// ---- DUTs/METS/Device/Scanner/Hand Scanner/ST_SCANNER_USBConfig.TcDUT
TYPE ST_SCANNER_USBConfig :
STRUCT
	bEnabled					: BOOL;										(* Enable HandScanner *)
	sScannerName				: STRING	:= 'USB';
	bReset					: BOOL;										(* Reset HandScanner *)
	nScannerPosition			: UINT;										(* Array position used in the camera configs.  This allows the HMi to display the handscanner stuff as a microscan camera *)
	sComPort					: STRING(5) := 'COM3';									(* COM port type*)
	nBaudRate				: UINT:= 9600;								(* Baud rate for scanner. 2 = 1200, 3=2400, 4=4800, 5=9600, 6=19200, 7=38400, 8=57600, 9=115200 - Default baudrate for hand sanner sick1910i *)          								 (* 1  *)
	tRXTimeOut				: TIME := T#0ms;
	nPackPerOuter				: INT := 20;
END_STRUCT
END_TYPE

// ---- DUTs/METS/Device/Scanner/NewModel/ST_SCANNER_Ctrl.TcDUT
TYPE ST_SCANNER_Ctrl :    //ST_SCANNER_CameraMap
STRUCT
	bProcessNewCode		: BOOL;
	bTCPTrigger			: BOOL;
	bManualTrigger		: BOOL;
	bResetStats			: BOOL;	
	
	stOptions			: ST_SCANNER_Options;
	stCameraMap			: ST_SCANNER_CtrlMapping;
END_STRUCT
END_TYPE

// ---- DUTs/METS/Device/Scanner/NewModel/ST_SCANNER_CtrlOptions.TcDUT
TYPE ST_SCANNER_CtrlOptions :
STRUCT
	eScannerType			: E_SCANNER_DeviceType;
	nImageBuffer			: INT;
	(*nSequenceProgs		: BYTE;*)
	bUseExternalLight		: BOOL;
	nExpectedResp			: INT;
END_STRUCT
END_TYPE

// ---- DUTs/METS/Device/Scanner/NewModel/ST_SCANNER_IN.TcDUT
TYPE ST_SCANNER_IN :
STRUCT
	stTriggerID				: ST_SCANNER_TriggerID;	(* trigger ID data, will be returned in sImageData to allow trigger and response to be aligned *)
	stManualStatus			: ST_SCANNER_ManualStatus;
	
END_STRUCT
END_TYPE

// ---- DUTs/METS/Device/Scanner/ST_SCANNER.TcDUT
TYPE ST_SCANNER :
STRUCT
	bReady							: BOOL;
	nState							: BYTE;
	bLastBarcodeValid					: BOOL;
(**)	strLastCodeRead					: T_MaxString;
(**)	strLastBarcode						: STRING(253);	(*zenon*)
	strCurrentCodeRead					: T_MaxString;
	aLast10CodesRead					: ARRAY[1..10]  OF T_MaxString;
	strLastStatus						: T_MaxString;
	nTriggerCounter					: UDINT;
	sManualCtrlScanner					: ST_SCANNER_ManualCtrl;
(**)(*	sSStats							: ST_SCANNER_Statistics;*)
	sScannerOpState					: ST_SCANNER_OpState;
	sImageData						: ST_SCANNER_ImageData;
	bEnableActive						: BOOL;
	nActiveProgram					: BYTE;
	bAcceptTrigger						: BOOL;
	sTriggerID							: ST_SCANNER_TriggerID;
	eSocketState						: E_SocketConnectionState;
	sReadPerformance					: ST_SCANNER_Performance;
END_STRUCT
END_TYPE

// ---- DUTs/METS/Device/Scanner/ST_SCANNER_ApplicationIdentifier.TcDUT
TYPE ST_SCANNER_ApplicationIdentifier :
STRUCT
	strAI		: STRING(4);
	bFixed		: BOOL;
	nLength		: UINT;
END_STRUCT
END_TYPE

// ---- DUTs/METS/Device/Scanner/ST_SCANNER_CameraMap.TcDUT
TYPE ST_SCANNER_CameraMap :
STRUCT
	nIndex				: INT;
	nReqProgram			: BYTE;
	stOptions				: ST_SCANNER_Options;
	aPackPos				: ARRAY[1..5, 1..cMAX_CAMERA_PROG_NUMBER] OF BYTE;
	aTargetBuffer			: ARRAY[1..5] OF BYTE;

END_STRUCT
END_TYPE

// ---- DUTs/METS/Device/Scanner/ST_SCANNER_CodeData.TcDUT
TYPE ST_SCANNER_CodeData :
STRUCT
	nScannerIndex			: INT;			(* scanner index when an array of scanners is used *)
	strDataString			: T_MaxString;	(* data string read from code *)
	eCodeType			: E_SCANNER_CodeType;	(* code type *)
	fOverallGrade			: LREAL;		(* overall grade of code *)
	fXPos				: LREAL;		(* X position of centre of code *)
	fYPos				: LREAL;		(* Y position of centre of code *)
	fAngle				: LREAL;		(* angle of code *)
	fCellSize				: LREAL;		(* cell size *)
	fSymbolContrast		: LREAL;		(* symbol contrast *)
	nEvaluation			: INT;			(* general code quality evaluatio*)
	fUnusedErrCorr			: LREAL;		(* unused error correction *)
	nProgramNo			: BYTE;			(* program number *)
END_STRUCT
END_TYPE

// ---- DUTs/METS/Device/Scanner/ST_SCANNER_Config.TcDUT
TYPE ST_SCANNER_Config :
STRUCT
	sDeviceName				: STRING(30) := 'Camera';
	bDisableCameraUse		: BOOL;
	aCameraWarningLevel		: INT := 90;
	stCameraIP					: ST_TCPIP_AddressPort;
	tTimeOut					: TIME := t#3s;
	eCameraVendor			: E_SCANNER_Vendor;
	bDontParseAsGS1			: BOOL;

	eScannerType			: E_SCANNER_DeviceType;
	eExpectedType			: E_SCANNER_CodeType;
	bUseExternalLight		: BOOL;
	nLightingIntensity		: INT;
	nDisplayDelayConfig	: BOOL;

	nImageBuffer			: INT := 1;
	nExpectedResp			: INT := 1;
END_STRUCT
END_TYPE

// ---- DUTs/METS/Device/Scanner/ST_SCANNER_Evaluation.TcDUT
TYPE ST_SCANNER_Evaluation :
STRUCT
	nTotalReads			: UDINT;
	nReadCodes			: UDINT;
	nNOKCodes			: UDINT;

	nGoodCodes			: UDINT;
	nFairCodes			: UDINT;
	nPoorCodes			: UDINT;

	fReadEfficiency			: LREAL;
	fNOKEfficiency			: LREAL;

	fGoodEfficiency		: LREAL;
	fFairEfficiency			: LREAL;
	fPoorEfficiency			: LREAL;

END_STRUCT
END_TYPE

// ---- DUTs/METS/Device/Scanner/ST_SCANNER_ImageData.TcDUT
TYPE ST_SCANNER_ImageData :
STRUCT
	nCodesRead		: INT;
	tScanTime		: TIME;		(* image cycle time (including image acquisition time and decode time) *)
	sStatus			: T_MaxString;
	stTriggerID		: ST_SCANNER_TriggerID;
	aCodeData		: ARRAY[1..cMAX_CAMERA_PROG_NUMBER] OF ST_SCANNER_CodeData;
END_STRUCT
END_TYPE

// ---- DUTs/METS/Device/Scanner/ST_SCANNER_ManualCtrl.TcDUT
TYPE ST_SCANNER_ManualCtrl :
STRUCT
	bManualTrigger		: BOOL;		(*zenon*)
	bConfigure			: BOOL;		(*zenon*)
	bBrowseLive			: BOOL;		(*zenon*)
	bBrowseDiag			: BOOL;		(*zenon*)
	bResetStats			: BOOL;		(*zenon*)
END_STRUCT
END_TYPE

// ---- DUTs/METS/Device/Scanner/ST_SCANNER_OpState.TcDUT
TYPE ST_SCANNER_OpState :
STRUCT
	bReady				: BOOL;
	nActiveProgram		: BYTE;
	bAcceptTrigger		: BOOL;
	bCodeChangeActive	: BOOL;
	nActiveTriggers		: INT;
	nExpectedResp			: INT;
	tAcquisitionTime	: TIME;
	nStatusByte			: BYTE;
	nErrorCode			: UDINT;
	nOpState			: BYTE;
END_STRUCT
END_TYPE

// ---- DUTs/METS/Device/Scanner/ST_SCANNER_Options.TcDUT
TYPE ST_SCANNER_Options :
STRUCT
	eScannerType			: E_SCANNER_DeviceType;
	nImageBuffer			: INT;
	(*nSequenceProgs		: BYTE;*)
	bUseExternalLight		: BOOL;
	nExpectedResp			: INT;
END_STRUCT
END_TYPE

// ---- DUTs/METS/Device/Scanner/ST_SCANNER_Performance.TcDUT
TYPE ST_SCANNER_Performance :
STRUCT
	tLastDiff : TIME;
	tAverageDiff : TIME;
	arrTimeDiff : ARRAY[0..9] OF TIME;
END_STRUCT
END_TYPE

// ---- DUTs/METS/Device/Scanner/ST_SCANNER_Statistics.TcDUT
TYPE ST_SCANNER_Statistics :
STRUCT
	nTotalReads			: UDINT;
	nValidCodes			: UDINT;
	nInvalidCodes			: UDINT;
	nDuplicateCodes		: UDINT;
	nNoCodeFound		: UDINT;
END_STRUCT
END_TYPE

// ---- DUTs/METS/Device/Scanner/ST_SCANNER_TriggerID.TcDUT
TYPE ST_SCANNER_TriggerID :
STRUCT
	nTriggerID			: UDINT;
	nScanNo				: INT := 1;
	nScannerIndex		: INT := 1;
END_STRUCT
END_TYPE

// ---- DUTs/METS/Files/E_FILE_CtrlState.TcDUT
TYPE E_FILE_CtrlState :
(
	E_CX_FILEIDLE,
	E_CX_FILEOPEN,
	E_CX_FILESEEK,
	E_CX_FILEREAD,
	E_CX_FILEWRITE,
	E_CX_FILECLOSE,
	E_CX_FILEDONE
);
END_TYPE

// ---- DUTs/METS/Files/E_FILE_DeleteOldFilesState.TcDUT
TYPE E_FILE_DeleteOldFilesState :
(
	E_OLDFILE_IDLE,
	E_OLDFILE_CURRENTTIME,
	E_OLDFILE_FILELIST1,
	E_OLDFILE_DELETEFILELIST1,
	E_OLDFILE_FILELIST2,
	E_OLDFILE_DELETEFILELIST2,
	E_OLDFILE_ABORTFILELIST,
	E_OLDFILE_FINDFOLDER,
	E_OLDFILE_FINDFILE,
	E_OLDFILE_DELETEFOLDER,
	E_OLDFILE_DELETEFILE,
	E_OLDFILE_DONE
);
END_TYPE

// ---- DUTs/METS/Files/E_FILE_State.TcDUT
TYPE E_FILE_State :
(
	E_FILE_IDLE,
	E_FILE_GETSIZE,
	E_FILE_OPEN,
	E_FILE_OPEN2,
	E_FILE_READ,
	E_FILE_READ2,
	E_FILE_WRITE,
	E_FILE_CLOSE,
	E_FILE_CLOSE2,
	E_FILE_COPY,
	E_FILE_COMPARE,
	E_FILE_ABORT,
	E_FILE_DELETE,
	E_FILE_MOVE,
	E_FILE_CHECKIFEXISTS,
	E_FILE_SEEK,
	E_FILE_FINDFILE,
	E_FILE_NEXTFILE,
	E_FILE_CLOSELIST,
	E_FILE_DONE
);
END_TYPE

// ---- DUTs/METS/Files/ST_FILE_WriteFileStatistic.TcDUT
TYPE ST_FILE_WriteFileStatistic :
STRUCT
	nTotalFilesWritten				: UDINT;
	nGoodFilesWritten				: UDINT;
	nBadFilesWritten				: UDINT;
	nFileWriteErrors				: UDINT;

	nTotalFilesVerified				: UDINT;
	nEmptyFilesVerified				: UDINT;
	nSizeErrorsVerified				: UDINT;
	nGoodFilesVerified				: UDINT;
	nFileVerifyNotFound			: UDINT;
	nFileVerifyErrors				: UDINT;
END_STRUCT
END_TYPE

// ---- DUTs/METS/HMI/Device Manual Control/ST_HMI_AxisCtrl.TcDUT
TYPE ST_HMI_AxisCtrl :
STRUCT
	stReqEanble		: ST_HMI_Buttons;
	stReqReset		: ST_HMI_Buttons;
	stReqPositioning	: ST_HMI_Buttons;	(*Button start positioning manual mode*)
	stRelease			: ST_HMI_Buttons;

	stReqJogFwd			: ST_HMI_Buttons;		(* set TRUE to jog forwards *)
	stReqJogRev			: ST_HMI_Buttons;		(* set TRUE to jog reverse *)
	fJogVelocity			: LREAL;	(* jog velocity (does not take effect if jog is in progress *)

	eMotionType		: E_AXIS_MotionType;

	fDistance			: LREAL;	(*target relative position*)
	fPosition			: LREAL;	(*target absolute position*)
	fVelocity			: LREAL;	(* target velocity *)
	bStopAtPos		: BOOL;	(* set TRUE to stop at specified pos, set FALSE to stop immediately *)
	fStopPos			: LREAL;	(* target modulo stop position *)

	(*eMotionState 		: MC_AxisStates;*)

END_STRUCT
END_TYPE

// ---- DUTs/METS/HMI/Device Manual Control/ST_HMI_G120Ctrl.TcDUT
TYPE ST_HMI_G120Ctrl :
STRUCT
	stRun				: ST_HMI_Buttons;
	stReset				: ST_HMI_Buttons;
	nSpeedHz 			: UINT;
	stInvertDirection	: ST_HMI_Buttons;
END_STRUCT
END_TYPE

// ---- DUTs/METS/HMI/Device Manual Control/ST_HMI_PrinterCtrl.TcDUT
TYPE ST_HMI_PrinterCtrl :
STRUCT
	stPrinterSelect		: ST_HMI_Buttons;
	stPrintLabel		: ST_HMI_Buttons;
	stApplyLabel		: ST_HMI_Buttons;	(*Button start positioning manual mode*)
	stPrinterReset		: ST_HMI_Buttons;

END_STRUCT
END_TYPE

// ---- DUTs/METS/HMI/Device Status/E_HMI_DriveStatus.TcDUT
TYPE E_HMI_DriveStatus :
(
	E_DRIVE_UNKNOWN := 0,
	E_DRIVE_SPOPPED := 1,
	E_DRIVE_RUNING := 2,
	E_DRIVE_ERROR := 3
);
END_TYPE

// ---- DUTs/METS/HMI/Device Status/ST_HMI_AxisStatus.TcDUT
//{warning 'CONVERSION MESSAGE: This text contained unprintable characters, that have been deleted'.}
TYPE ST_HMI_AxisStatus :
STRUCT

(* read only *)

	eMotionState 		: MC_AxisStates;

	bInitOK				: BOOL;
	bEnabled			: BOOL;
	bHomeActive			: BOOL;
	bVeloActive			: BOOL;
	bRelativeActive		: BOOL;
	bAbsoluteActive		: BOOL;
	bJogActive			: BOOL;


	bOperational 				: BOOL;
	bHasJob						: BOOL;
	bInTargetPosition 			: BOOL;
	bInPositionRange 			: BOOL;
	bHomed 						: BOOL;
	bHomingBusy 				: BOOL;
	bMovingPositiveDirection 	: BOOL;
	bMovingNegativeDirection	: BOOL;
	bNotMoving 					: BOOL;

	bError 						: BOOL;
	nErrorId 					: UDINT;

	fActualPosition 			: LREAL;
	fActualVelocity 			: LREAL;
	fSetpointPosition 			: LREAL;


END_STRUCT
END_TYPE

// ---- DUTs/METS/HMI/Device Status/ST_HMI_CylinderStatus.TcDUT
TYPE ST_HMI_CylinderStatus :
STRUCT

(* read only *)
	bDeviceDisable			: BOOL;
	bMoveNotAllowed			: BOOL;

	bErrorPosition				: BOOL;
	bInPosition				: BOOL;
	bHomePosition				: BOOL;

	bCylinderInRetractedPosition	: BOOL;
	bCylinderInExtendedPosition	: BOOL;
	bCylinderIsRetracting		: BOOL;
	bCylinderIsExtending		: BOOL;

	stTagID					: ST_CYLINDER_TagID;

END_STRUCT
END_TYPE

// ---- DUTs/METS/HMI/Device Status/ST_HMI_HoneywellStatus.TcDUT
TYPE ST_HMI_HoneywellStatus :
STRUCT

(* read only *)
	bHandScanerPortOK			: BOOL;
	bHandScannerBaudrateOK	: BOOL;
	sLastScannerBarcode		: T_MaxString;

END_STRUCT
END_TYPE

// ---- DUTs/METS/HMI/Device Status/ST_HMI_PrinterStatus.TcDUT
TYPE ST_HMI_PrinterStatus :
STRUCT
	sPrinterName					: STRING(30);
(* read only *)
	bPrinterReady					: BOOL;
	bActivePrinter					: BOOL;
	bPrinterInService				: BOOL;		(*printer Avalable*)
	bPrinterSelected				: BOOL;
	bDataReady					: BOOL;
	bHomePosition				: BOOL;
	bLabelPrinted					: BOOL;
	bReadyToApply				: BOOL;
	bApplyDone					: BOOL;
	bSummaryWarning				: BOOL;
	bPrinterError					: BOOL;

	Q								: ST_PRINTER_OUT;

END_STRUCT
END_TYPE

// ---- DUTs/METS/HMI/HMIQueue/ST_HMI_CAC_Data.TcDUT
TYPE ST_HMI_CAC_Data :
STRUCT
	sBarcode 				: T_CASE_Barcode;
	(*sCaseIDCode			: STRING(10);
	sProductionDate			: STRING(10);
	sProductionTime			: STRING(8);
	sCaseRejectCode			: T_MaxString;		(* blank and not included in CAC files for valid cases *)*)
	nNumberOfOuters			: INT;
	nNumberOfPacks			: INT;
	aOuter					: ARRAY[1..cMAX_HMI_OUTERS_PER_CASE] OF ST_HMI_OAC_Data;
END_STRUCT
END_TYPE

// ---- DUTs/METS/HMI/HMIQueue/ST_HMI_CaseVerifiedCode.TcDUT
TYPE ST_HMI_CaseVerifiedCode :
STRUCT
	sCaseIDCode				: STRING(10);
	sProductionDate			: STRING(10);
	sProductionTime			: STRING(8);
END_STRUCT
END_TYPE

// ---- DUTs/METS/HMI/HMIQueue/ST_HMI_CASE_CaseQueue.TcDUT
TYPE ST_HMI_CASE_CaseQueue :
STRUCT
	aCACData		: ARRAY[1..cMAX_CASE_QUEUE] OF ST_HMI_CAC_Data;	(* array of CAC data *)
END_STRUCT
END_TYPE

// ---- DUTs/METS/HMI/HMIQueue/ST_HMI_OAC_Data.TcDUT
TYPE ST_HMI_OAC_Data :
STRUCT
	sBarcode				: T_OUTER_Barcode;
	aPackCode				: ARRAY[1..cMAX_HMI_PACKS_PER_OUTER] OF T_HMI_PACK_Barcode;
END_STRUCT
END_TYPE

// ---- DUTs/METS/HMI/HMIQueue/ST_HMI_OCV_Data.TcDUT
TYPE ST_HMI_OCV_Data :
STRUCT
	sPackCode			: T_PACK_Barcode;
	nPackStatus		: BYTE;
END_STRUCT
END_TYPE

// ---- DUTs/METS/HMI/HMIQueue/ST_HMI_OuterStatus.TcDUT
TYPE ST_HMI_OuterStatus :
STRUCT
	sBarcode						: T_OUTER_Barcode;

	sOuterRejectCode				:  T_RejectCode;
	nOuterRejectID					:  UINT;

	aAggregationCodes			: ARRAY[1..2] OF T_PACK_Barcode;
	aAggregationCodesPosition	: ARRAY[1..2] OF INT;

	aPackRejectCode				: ARRAY[1..cMAX_HMI_PACKS_PER_OUTER] OF T_RejectCode;
	aPackRejectID					: ARRAY[1..cMAX_HMI_PACKS_PER_OUTER] OF INT;

	sProductionDate				: STRING(10);
	sProductionTime				: STRING(8);

	aPackCode						: ARRAY[1..cMAX_HMI_PACKS_PER_OUTER] OF T_PACK_Barcode;
	aOACPackStatus				: ARRAY[1..cMAX_HMI_PACKS_PER_OUTER] OF BYTE;	(* OAC pack code status *)

	nNumberOfPacks				: INT;
	nAcceptanceLevel				: INT;
	nNumberOfLinkedPacks		: INT;
	nMaxOuterStatusQueue		: INT;

END_STRUCT
END_TYPE

// ---- DUTs/METS/HMI/HMIQueue/ST_HMI_PLAS_Queue.TcDUT
TYPE ST_HMI_PLAS_Queue :
STRUCT
(*Pack Infeed queue*)
	nInfeedIndex					: INT;				(* number of Outers in queue *)
	aPackInfeedQueue				: ARRAY[1..cMAX_HMI_PACK_INFEED_QUEUE] OF T_HMI_PACK_Barcode; (* pack infeed queue + status (999)*)

(*Pack Buffer intermediat queue*)
	aBufferQueue					: ARRAY[1..cMAX_HMI_PACK_INFEED_QUEUE] OF T_HMI_PACK_Barcode; (* intermediat pack queue + status (999)*)

(*OCV Data*)
	sProductionDate				: STRING(10);
	sProductionTime				: STRING(8);

	aOCVData						: ARRAY[1..cMAX_HMI_PACKS_PER_OUTER] OF T_HMI_PACK_Barcode; (* pack queue + status (999)*)

	nNumberOfPacks				: INT;
	nAcceptanceLevel				: INT;
	nNumberOfLinkedPacks		: INT;
	nMaxPackPerOuter				: INT; (*real number of codes*)

END_STRUCT
END_TYPE

// ---- DUTs/METS/HMI/ST_HMI_Buttons.TcDUT
TYPE ST_HMI_Buttons :
STRUCT

	bButtonState			: 	BOOL;
	bButtonRisingEdge		:	BOOL;
   	bButtonFallingEdge		:	BOOL;
	(*nChangeLogID			: 	INT;*)


(*	bStartButtonRisingEdge		:	BOOL;
   	bStartButtonFallingEdge		:	BOOL;
    	bResetButtonRisingEdge		:	BOOL;
    	bResetButtonFallingEdge		:	BOOL;
    	bStopButtonRisingEdge		:	BOOL;
    	bStopButtonFallingEdge		:	BOOL;*)
END_STRUCT
END_TYPE

// ---- DUTs/METS/HMI/ST_HMI_StationStatus.TcDUT
TYPE ST_HMI_StationStatus :
STRUCT

	bSeqAbort					: BOOL;		(**)
	bSeqIsHoming				: BOOL;
	bSeqInProgress				: BOOL;		(**)
	bSeqComplete				: BOOL;		(**)
	bSeqError					: BOOL;
	nSeqErrorID					: UDINT;

	bStationHomed				: BOOL;		(**)
	bStationNotMoving			: BOOL;		(**)



END_STRUCT
END_TYPE

// ---- DUTs/METS/HMI/ST_HMI_Visualisation.TcDUT
TYPE ST_HMI_Visualisation:
STRUCT
	(*Test outputs*)
(*	bEnableForcingOutputs			: BOOL;

	bForceEUCAMachineRun_STCP		: BOOL;	(*to set qb82KF1_1_EUCAMachineRun*)
	bForceCaseValidationOK_STCP		: BOOL;	(*to set qb82KF1_5_CaseValidationOK*)
	bForceOuterValidationOK_STCP	: BOOL;	(*to set qb82KF1_2_OuterValidationOK*)
	bForceLabellerInhibit_STL		: BOOL;	(*to set qb82KF1_3_LabellerInhibit_STL*)
	bForceTPDMachineRun			: BOOL;	(*to set qb482KF1_4_TPDMachineRun*)
	bForceSpare					: BOOL;
*)

	(*Update PCM*)
	bEnableUpdatePCM				: BOOL;

	strLastRetailSKU 				: T_CodeRSKU;
	strLastProductionOrder			: T_CodePO;
	strLastBatchNumber				: T_CodeBATCH;

	strLastPackGTIN 				: T_CodeGTIN;
	strLastOuterGTIN 				: T_CodeGTIN;
	strLastCaseGTIN 				: T_CodeGTIN;

END_STRUCT
END_TYPE

// ---- DUTs/METS/KPI/ST_KPI_CasePackerSignals.TcDUT
TYPE ST_KPI_CasePackerSignals :
STRUCT
	nSensor			: UDINT;
	nMachine		: UDINT;
	nPLC			: UDINT;

END_STRUCT
END_TYPE

// ---- DUTs/METS/KPI/ST_KPI_CodePos.TcDUT
TYPE ST_KPI_CodePos :
STRUCT
	ReadOK				: UDINT;
	Efficiency			: LREAL;
END_STRUCT
END_TYPE

// ---- DUTs/METS/KPI/ST_KPI_InspectionEfficency.TcDUT
TYPE ST_KPI_InspectionEfficency :
STRUCT
	ProcessedTotal			: UDINT;
	ProcessedSuccessful		: UDINT;
	ProcessedRejected		: UDINT;
	ProcessedEfficiency		: LREAL;
END_STRUCT
END_TYPE

// ---- DUTs/METS/KPI/ST_KPI_ItemsProduced.TcDUT
TYPE ST_KPI_ItemsProduced :
STRUCT
	Total					: UDINT;
	Passed				: UDINT;
	Rejected				: UDINT;
	Efficiency				: LREAL;
	CreatedFiles			: UDINT;
	WarningLevel			: REAL := 99.75;
	AlarmLevel			: REAL := 99.50;
END_STRUCT
END_TYPE

// ---- DUTs/METS/KPI/ST_KPI_OCVFile.TcDUT
TYPE ST_KPI_OCVFile :
STRUCT
	nOCVFiles					: UDINT;
	nOuterStoredInOCV				: UDINT;
	nLinkedPackInOCV				: UDINT;
	nOCVWriteErrorCounter			: UDINT;
END_STRUCT
END_TYPE

// ---- DUTs/METS/KPI/ST_KPI_OutersProcessing.TcDUT
TYPE ST_KPI_OutersProcessing :
STRUCT
	AtPackAggregCameras	: UDINT;
	AtConfimrationCamera 	: UDINT;
	AtValidationCamera		: UDINT;
END_STRUCT
END_TYPE

// ---- DUTs/METS/KPI/ST_KPI_OutersProduced.TcDUT
TYPE ST_KPI_OutersProduced :
STRUCT
	Total					: UDINT;
	Passed				: UDINT;
	Rejected				: UDINT;
	Efficiency				: LREAL;
END_STRUCT
END_TYPE

// ---- DUTs/METS/LogData/E_LOG_Handler.TcDUT
{attribute 'qualified_only'}
TYPE E_LOG_Handler :
(
	
(**************** Keep in mind limited number of E_NUM elements (array of FB handlers) fixed size to 256 ******************)
		
(* FSS connection logs *)
		OKCONECCTIONTOFSS,
		LOSTCONECCTIONTOFSS,
		
		(* Doors logs*)
		DOOROPENZONE1,
		DOOROPENZONE2,
		MASTERLISTDOOR,
		AGGREGATIONDOOR,
		PACKWRAPPERDOOR,
		
(* Control buttons logs*)
		STARTBUTTONPRESSED,
		STOPBUTTONPRESSED,
		RESETBUTTONPRESSED,
		
(* Machines not running status logs *)
		EUCANOTRUNNINGPT,
		EUCANOTRUNNINGCT,
		TPDNOTRUNNINGPT,
		TPDNOTRUNNINGCT,	
		EXTNOTRUNNINGPT,
		EXTNOTRUNNINGCT,
		
(* Machines state changed *)
		MACHINESTATEPT,
		MACHINESTATECT,
		
(**************** PACK AGGREGATION MODE ****************)		
		
(*PAOL SEQUENCE - 2CAM_METSONE*)				
		PAOL2CAMPACKAGGTRIG,		
		PAOL2CAMCAM1,		
		PAOL2CAMCAM2,
		PAOL2CAMPA1ADDED,
		PAOL2CAMPA2ADDED,	
		
(*PAOL SEQUENCE - 3CAM_LIHTBOX*)
		PAOL3CAMPA1ADDED,		
		PAOL3CAMPA2ADDED,
		PAOL3CAMPA3ADDED,
		
(*PLAS SEQUENCE - T01*)
		T01CAMAGG1,
		T01CAMAGG2,		
		T01CAMAGGTRIG,
		T01STACKERTRIG,
		T01AGGITEM,
		T01AGGADDED,
		T01WRAPPER1REJECT,
				
(*PLAS SEQUENCE - T02*)
		T02CAMAGG1,
		T02CAMAGG2,
		T02CAMAGGTRIG,
		T02STACKERTRIG,
		T02CAMINTERTRIG,
		T02CAMINTER,
		T02INTERQUEUE,
		T02AGGITEM,
		T02AGGADDED,
		T02WRAPPER1REJECT,
		
(*PLAS SEQUENCE - T03*)
		T03CAMAGG,
		T03CAMAGGTRIG,
		T03CAMCONFTRIG,
		T03CAMINTERTRIG,
		T03CAMINTER,
		T03INTERQUEUE,
		T03CAMCON,
		T03PACKINDEX,
		T03MOVEDTOOCV,
		T03WRAPPERREJECT,
		
(*PLAS SEQUENCE - T04*)		
		T04CAMAGG,
		T04CAMAGGTRIG,	
		T04CAMCONFTRIG,
		T04CAMINTERTRIG,
		T04CAMINTER,
		T04INTERQUEUE,
		T04CAMCON,
		T04PACKINDEX,
		T04MOVEDTOOCV,
		T04WRAPPERREJECT,
		
(**************** PACK AGGREGATION MODE ****************)
		
(* OCV logs *)
		STACKOUTOFSEQ,
		LASTOCVCONTENT,
		
(* OAC logs *)
		LASTOACCONTENT,
		
(* Printers comands *)
		LASTPRINTER01COMMAND,
		LASTPRINTER02COMMAND,
		LASTPRINTER03COMMAND,
		LASTPRINTER04COMMAND,
		LASTPRINTER05COMMAND,
		LASTPRINTER06COMMAND,
		
(* Case Packer Sequence logs *)
		OUTERCOMPLETE,
		ROWCOMPLETE,
		LAYERCOMPLETE,
		INTERMEDIATECOMPLETE,
		CASECOMPLETE,		
		CASEDISCHARGERT,
		CASEDISCHARGEFT,
		CASELABELVALIDATION,
		
(* Cameras timeout logs *)
		OUTERAGGREGATIONCODE,
		
(* Data move/handeling status logs*)
		ROWCOMPLETECODES,
		LAYERCOMPLETECODES,
		FINALISECASECONTENTCODES,
		
(* Data LogIn DB logs*) (* NOT INTUITIVE NAMES - to be changed ?? *)
		INTERPUSHOVERWIRTTEN,
		CASECOMPLETEOVERWITTEN,
		CASEDISCHARGEOVERWRITTEN,
		
(* Rejects handling logs *)
		REJECTEDBYCASEPACKER,
		
(* Case events logs *)
		CASELABELCODE,
		MCCREATEDEVENT,
		CASEVALIDATIONRT,
		CASEVALIDATIONFT,
		
(* Data files write error logs *)
		OCVWRITEERROR,
		OACWRITEERROR,
		CACWRITEERROR,
		CHMWRITEERROR,
		
(* Master List status logs *)
		MLFILLINSTATUS,
		MLSTATUS,
		MLRESOTRESTATUS,
		//E_LOG_WRAPPERREJECT1,
		WRAPPERREJECT2
		
);
END_TYPE

// ---- DUTs/METS/LogData/ST_LOG_Alarms.TcDUT
TYPE ST_LOG_Alarms :
STRUCT

	nAlarmCounter				: UINT;
	sTotalAlarmTime				: T_TimeLog;
	sMaxAlarmTime				: T_TimeLog;
	stMaxAlarmTimeStamp			: TIMESTRUCT;

END_STRUCT
END_TYPE

// ---- DUTs/METS/LogData/ST_LOG_EventData.TcDUT
TYPE ST_LOG_EventData :
STRUCT
	bEnable					: BOOL;
	nCounter				: UDINT;
	sTimeStamp				: STRING;
	nImageByte				: UINT;
	aDataLogImage			: ARRAY[0..65000] OF BYTE;
	nMaxImageArraySize		: UINT := 65000 ;
	nControlSize			: UINT;
	bBufferOverflow			: BOOL;
END_STRUCT
END_TYPE

// ---- DUTs/METS/LogData/ST_LOG_FileWriteError.TcDUT
TYPE ST_LOG_FileWriteError :
STRUCT
	nWriteErrorID			: UDINT;
	sTimeStamp				: STRING;
	strFileName				: T_MaxString;
END_STRUCT
END_TYPE

// ---- DUTs/METS/LogData/ST_LOG_MachineState.TcDUT
TYPE ST_LOG_MachineState :
STRUCT

	sPowerUp					: T_TimeLog;
	sImmediateStopped			: T_TimeLog;
	sMachineInError				: T_TimeLog;
	sSystemInitialising			: T_TimeLog;
	sSystemManual				: T_TimeLog;
	sSystemReadytoStart			: T_TimeLog;
	sStopping					: T_TimeLog;
	sSystemRunning				: T_TimeLog;
	sMachineWaitingForProduct	: T_TimeLog;
	sConveyorModeActive			: T_TimeLog;
	sSystemConditionalRunning	: T_TimeLog;

END_STRUCT
END_TYPE

// ---- DUTs/METS/LogData/ST_LOG_WriteImageData.TcDUT
TYPE ST_LOG_WriteImageData :
STRUCT
	aLogPT			: ARRAY[0..65000] OF BYTE;
	aLogML			: ARRAY[0..65000] OF BYTE;
	aLogOT			: ARRAY[0..65000] OF BYTE;
	aLogCT			: ARRAY[0..65000] OF BYTE;
END_STRUCT
END_TYPE

// ---- DUTs/METS/NV Data/ST_NOVRAM_METS_Cameras.TcDUT
TYPE ST_NOVRAM_METS_Cameras :
STRUCT
	MachineID					: ST_SYSTEM_MachineID;
	StartDateTime					: T_ISO8601Time;
	CodingAndTrackingMode			: INT;

	aCameraEvaluation				: ARRAY[1..cMAX_CAMERA_NUMBER] OF ST_SCANNER_Evaluation;

	(*CameraPackEval				: ARRAY[1..6] OF ST_SCANNER_Evaluation;
	CameraConfirmEval				: ARRAY[1..2] OF ST_SCANNER_Evaluation;
	CameraOuterValidEval			: ST_SCANNER_Evaluation;
	CameraOuterAggregEval			: ST_SCANNER_Evaluation;
	CameraCaseContentEval			: ST_SCANNER_Evaluation;
	CameraCaseLableEval			: ST_SCANNER_Evaluation;*)

END_STRUCT
END_TYPE

// ---- DUTs/METS/NV Data/ST_NOVRAM_METS_CaseInspactionLog.TcDUT
TYPE ST_NOVRAM_METS_CaseInspactionLog :
STRUCT

	MachineID						: ST_SYSTEM_MachineID;
	StartDateTime						: T_ISO8601Time;
	CodingAndTrackingMode				: INT;
	nPacksPerCase						: INT;			(* Amount Of  Packs per Case unit for current PCM *)
	nOutersPerCase					: INT;

	(*infeed conveyer*)
	nOuterProcessed					: UDINT;
	nOuterAggregated					: UDINT;
	nMasterListRestoredSuccessful		: UDINT;
	nMasterListRemoved				: UDINT;
	nQualityRejects					: UDINT;

	(*row validation*)
	nRowValidationIndexUnder			: UDINT;
	nRowValidationIndexOver			: UDINT;
	nRowValidationIndexCorrect			: UDINT;
	nRowValidationIndexNotFound		: UDINT;

	(*outer to case validation*)
	nOuterToCaseValidationIndexUnder		: UDINT;
	nOuterToCaseValidationIndexOver		: UDINT;
	nOuterToCaseValidationIndexCorrect	: UDINT;
	nOuterToCaseValidationIndexNoData	: UDINT;

	(*case validation*)
	nCaseValidationScanned				: UDINT;
	nCaseValidationCorrect				: UDINT;
	nCaseValidationCasePackerReject		: UDINT;
	nCaseValidationNoCaseLabel			: UDINT;


END_STRUCT
END_TYPE

// ---- DUTs/METS/NV Data/ST_NOVRAM_METS_DualInputs.TcDUT
TYPE ST_NOVRAM_METS_DualInputs :
STRUCT

	MachineID					: ST_SYSTEM_MachineID;
	StartDateTime					: T_ISO8601Time;
	CodingAndTrackingMode			: INT;

	RowComplete			:	ST_KPI_CasePackerSignals;
	LayerComplete			:	ST_KPI_CasePackerSignals;
	CaseComplete			:	ST_KPI_CasePackerSignals;
	CaseDischarged		:	ST_KPI_CasePackerSignals;
	CaseLabelValidation		:	ST_KPI_CasePackerSignals;


END_STRUCT
END_TYPE

// ---- DUTs/METS/NV Data/ST_NOVRAM_METS_Inspection.TcDUT
TYPE ST_NOVRAM_METS_Inspection :
STRUCT
	MachineID					: ST_SYSTEM_MachineID;
	StartDateTime					: T_ISO8601Time;
	CodingAndTrackingMode			: INT;
	AcceptanceLevel				: INT;
	PacksPerOuter					: INT;
	OutersProcessing				: ST_KPI_OutersProcessing;
	OCVFileEfficiency				: ST_KPI_OCVFile;

	PacksRead					: ARRAY[0..cMAX_PACKS_PER_OUTER] OF UDINT;
	PackPosEfficiency				: ARRAY[1..cMAX_PACKS_PER_OUTER] OF ST_KPI_CodePos;

	PackAggregationEfficiency		: ST_KPI_InspectionEfficency;
	PackProduced					: ST_KPI_ItemsProduced;

	aConfirmCodeEfficiency			: ARRAY[1..2] OF ST_KPI_CodePos;
	PackConfirmationEfficiency		: ST_KPI_InspectionEfficency;
	aValidCodeEfficiency			: ARRAY[1..2] OF ST_KPI_CodePos;
	OuterValidationEfficiency			: ST_KPI_InspectionEfficency;

	OuterAggregationEfficiency		: ST_KPI_InspectionEfficency;
	OutersProduced				: ST_KPI_ItemsProduced;

	(*CaseContentValidEfficiency		: ST_KPI_InspectionEfficency;
	CaseLableValidEfficiency			: ST_KPI_InspectionEfficency;*)

	CaseAggregationEfficiency		: ST_KPI_InspectionEfficency;
	CaseProduced					: ST_KPI_ItemsProduced;


END_STRUCT
END_TYPE

// ---- DUTs/METS/Outers/E_OUTER_AgrregationState.TcDUT
TYPE E_OUTER_AgrregationState :
(
	E_OUTER_IDLE_OCV,
	E_OUTER_READ_OCV,
	E_OUTER_ERROR_OCV_READ,
	E_OUTER_BUILD_OAC_DATA,
	E_OUTER_DONE_OCV
);
END_TYPE

// ---- DUTs/METS/Outers/E_OUTER_State.TcDUT
TYPE E_OUTER_State :
(
	E_OUTER_IDLE,
	E_OUTER_SCAN,
	E_OUTER_VALIDATE,
	E_OUTER_CHECKPACKS,
	E_OUTER_KPI,
	E_OUTER_STATUS,
	E_OUTER_DBREQUEST,
	E_OUTER_DBRESPONSE,
	E_OUTER_BUILDXMLIMAGE,
	E_OUTER_WRITEXMLIMAGE,
	E_OUTER_WRITESECONDXMLIMAGE,
	E_OUTER_CREATEERRORFOLDER,
	E_OUTER_UPDATEDATA,
	E_OUTER_WRITEDATA,
	E_OUTER_DELETEFILE,
	E_OUTER_UPDATESTATUS,
	E_OUTER_FINDFILE,
	E_OUTER_READDATA,
	E_OUTER_UPDATEINFEEDQUEUE,
	E_OUTER_DELETECONVQUEUE,
	E_OUTER_DONE
);
END_TYPE

// ---- DUTs/METS/Outers/OAC/E_OAC_State.TcDUT
TYPE E_OAC_State :
(
	E_OAC_IDLE,
	E_OAC_HEADER,
	E_OAC_PACKDATA,
	E_OAC_MOVENAS,
	E_OAC_MOVELOCAL,
	E_OAC_VALIDATEOUTER,
	E_OAC_VALIDATEPACK,
	E_OAC_DBREQUEST,
	E_OAC_DBRESPONSE,
	E_OAC_READFILE,
	E_OAC_FINDFILE,
	E_OAC_DELETEFILE,
	E_OAC_DONE
);
END_TYPE

// ---- DUTs/METS/Outers/OAC/ST_OAC_Data.TcDUT
TYPE ST_OAC_Data :
STRUCT
	Barcode					: T_OUTER_Barcode;
	ProductionDate			: STRING(10);
	ProductionTime			: STRING(8);
	ProductionTimeOffset		: STRING(6);		(* time offset between system and UTC, '+1:00' means SystemTime = UTC + 1hr *)
	OuterTimeStamp				: T_ISO8601Time;
	PackTimeStamp				: T_ISO8601Time;
	RetailSKU					: T_CodeRSKU;
	OuterMachine				: ST_SYSTEM_MachineID;
	AggregationCodes			: ARRAY[1..2] OF T_PACK_Barcode; 		(* pack aggregation codes for CML *)
	OuterMasterListRestored		: BOOL;
	CodingAndTrackingMode		: INT;
	NumberOfPacks			: INT;
	AcceptanceLevel			: INT;
	NumberOfLinkedPacks		: INT;
	BatchNumber				: T_CodeBATCH;
	DataSource				: STRING(4);
	(*ProductCode5678			: STRING(4);*)
	OuterRejectCode			:  T_RejectCode;
	OuterRejectID				: UINT;
	OuterCodeStatus			: WORD;	(*16bits states *)
	PackCode					: ARRAY[1..cMAX_PACKS_PER_OUTER] OF T_PACK_Barcode;
	PackRejectCode			: ARRAY[1..cMAX_PACKS_PER_OUTER] OF T_RejectCode;
	PackRejectID				: ARRAY[1..cMAX_PACKS_PER_OUTER] OF UINT;
	PackCodeStatus			: ARRAY[1..cMAX_PACKS_PER_OUTER] OF WORD;			(*16bits states *)


(*OuterCodeStatus dcoding bits - concept.
b0		Outer Code - Database check performed
b1		Outer Code - Database error during check
b2		Outer Code - Found in database - DB validation OK
b3		Outer Code - has expired - result from DB check
b4 		Outer Code - Outer MasterList Restored
b5		Outer Code - Val Index error found
b6		Outer Code - OAC File Write Error
b7		Outer Code - OAC biuld form restored OCV
b8		Outer Code - Reserved of use in future
b9		Outer Code - Reserved of use in future
b10	Outer Code - Reserved of use in future
b11	Outer Code - Reserved of use in future
b12	Outer Code - Reserved of use in future
b13	Outer Code - Reserved of use in future
b14	Outer Code - Reserved of use in future
b15	Outer Code - Reserved of use in future

*)


(*	PackCodeStatus dcoding bits - concept.

b0	 	Pack code -  no readed.
b1 		Pack code - over-written.  2 different codes read for same Pack position
b2		Pack code - invalid GTIN/SerialLenght/CodeType/CodeLenght 
b3		Pack code - duplicate code found in one outer. Currentpack code contains data and matches another pack code. 
b4		Pack code - change status to indicate invalid packcode  in an accepted outer
b5		Pack code - valid code
b6		Pack code - packcode manually repaired ( restored manually by hand scanner), status used in arrErrorOuters only for HMI
b7		Pack code - Reserved of use in future 
b8	 	Pack code - Pack Data reanimated 
b9 		Pack code - restored by primary master list camera
b10   	Pack code - restored by secondary master list camera
b11	Pack code - pcakcode removed form the system (NCW)
b12	Pack code - Database check performed
b13	Pack code - Database error during check
b14 	Pack code - Pack found in database - DB validation OK
b15 	Pack code - has expired - result from DB check

*)
END_STRUCT
END_TYPE

// ---- DUTs/METS/Outers/SFLX/E_SIDEFLEX_UnitType.TcDUT
TYPE E_SIDEFLEX_UnitType :
(
	E_SIDEFLEX_UNKNOWN			:= 0,
	E_SIDEFLEX_2PROG				:= 1,
	E_SIDEFLEX_4PROG				:= 2
);
END_TYPE

// ---- DUTs/METS/Outers/SFLX/ST_SIDEFLEX_Offset.TcDUT
TYPE ST_SIDEFLEX_Offset :
STRUCT
	(*aTrigerPos		: ARRAY[0..cMAX_CAMERA_NUMBER] OF UDINT;*)

(*ONLY ONE OUTER AT THE TIME IN THIS RANGE FOR nCurrentPosition OR FOR nLeadingPosition*)
	nStartOuterAtLabellerPos	: UDINT;
	nEndOuterAtLabellerPos		: UDINT;

END_STRUCT
END_TYPE

// ---- DUTs/METS/Outers/SFLX/ST_SIDEFLEX_ProcessData.TcDUT
TYPE ST_SIDEFLEX_ProcessData :
STRUCT

	stOCVPackStatus			: ST_OUTER_Status;
	nCurrentPosition			: UDINT;
	nLeadingPosition			: UDINT;
	nTrailingPosition			: UDINT;
	nOuterLenght				: UDINT;

	bOCVUpdated				: BOOL;
	bOCVInvalid				: BOOL;

	bOuterAtLabeller			: BOOL;
	bApplyDone				: BOOL;
	bOuterCompleted			: BOOL;
	bOutrRejected				: BOOL;

END_STRUCT
END_TYPE

// ---- DUTs/METS/Outers/ST_OUTER_Status.TcDUT
TYPE ST_OUTER_Status :
STRUCT
	bOuterPresent		: BOOL;		(* TRUE = Outer present *)
	bLabelApplied		: BOOL;		(* TRUE = label has been printed and applied to Outer *)
	nTriggerID			: UDINT;	(* TriggerID value for scanners *)
	bOuterCodeValid		: BOOL;		(* TRUE = Outer code valid *)
	bPackCodesValid		: BOOL;		(* TRUE = Pack codes valid *)
	bQAReject			: BOOL;		(* TRUE = QA reject requested *)
	nStatus				: DWORD;
	sDataSourceTracker		: STRING(10);
	stOACData			: ST_OAC_Data;			(* OAC data for pack *)
	(*sOHMData		: ST_OHM_Data;		(*New OHM data structure*)*)
	aOACPackStatus		: ARRAY[1..cMAX_PACKS_PER_OUTER] OF BYTE;	(* OAC pack code status *)
	aPackSUPIResult		: ARRAY[1..cMAX_PACKS_PER_OUTER] OF DINT;	(* OAC pack code status *)
	aPackCodeFilledIn		: ARRAY[1..cMAX_PACKS_PER_OUTER] OF E_PACK_FilledInStatus;
	(*strAggregationCodes	: ARRAY[1..2] OF T_PACK_Barcode; 		(* pack aggregation codes for CML *)*)
	aPackCodes			: ARRAY[1..cMAX_PACKS_PER_OUTER] OF ST_PACK_CodeBuffer; 	(* primary and secondary buffers for pack codes *)
END_STRUCT
END_TYPE

// ---- DUTs/METS/Packs/E_OCV_CheckMode.TcDUT
TYPE E_OCV_CheckMode :
(
	E_OCV_CHECKOFF,
	E_OCV_PACKLEVEL,
	E_OCV_OUTERLEVEL

);
END_TYPE

// ---- DUTs/METS/Packs/E_OCV_State.TcDUT
TYPE E_OCV_State :
(
	E_OCV_IDLE,
	E_OCV_SCAN,

	E_OCV_DBREQUEST,
	E_OCV_DBRESPONSE,

	E_OCV_VALIDATENAME,
	E_OCV_VALIDATECONTENT,

	E_OCV_UPDATEDATA,
	E_OCV_WRITEDATA,
	E_OCV_MOVEFILE1,
	E_OCV_MOVEFILE2,

	E_OCV_FINDFILE,
	E_OCV_READFILE,
	E_OCV_READERRORFILE,
	E_OCV_DELETEFILE,

	E_OCV_UPDATESTATUS,
	E_OCV_DONE
);
END_TYPE

// ---- DUTs/METS/Packs/E_PACK_FilledInStatus.TcDUT
TYPE E_PACK_FilledInStatus :
(
	E_PACK_EMPTY := 0,
	E_PACK_SECONDARYMASTERLISTRESTORED :=1,
	E_PACK_PRIMARYMASTERLISTRESTORED :=2,
	E_PACK_CODEAGGREGATED :=3,
	E_PACK_CODERESTOREDFAILED := 4,
	E_PACK_CODEREMOVED :=5,
	E_PACK_CODERESTOREDCAC := 6,
	E_PACK_CODEOVERWRITTEN := 7
);
END_TYPE

// ---- DUTs/METS/Packs/E_PACK_ReadStep.TcDUT
TYPE E_PACK_ReadStep :
(
	E_DISARMED,

	E_RELAY_1,
	E_RELAY_235,
	E_RELAY_46,
	E_RELAY_78,

	E_2CAM_TRIG01,
	E_2CAM_TRIG02,
	E_2CAM_TRIG03,
	E_2CAM_TRIG04,
	E_2CAM_TRIG05,
	E_2CAM_TRIG06,
	E_2CAM_SEQDWELL

);
END_TYPE

// ---- DUTs/METS/Packs/E_PACK_State.TcDUT
TYPE E_PACK_State :
(
	E_PACK_IDLE,
	E_PACK_DBREQUEST,
	E_PACK_DBRESPONSE,
	E_PACK_CODEVALIDATION,
	E_PACK_DUPLICATECHEKC,
	E_PACK_VALIDECODEADD,
	E_PACK_INVLIDECODEADD,
	E_PACK_SCANINFEEDQUEUE,
	E_PACK_UPDATEINFEEDQUEUE,
	E_PACK_UPDATEOCVQUEUE,
	E_PACK_DONE

);
END_TYPE

// ---- DUTs/METS/Packs/ST_PACK_CodeBuffer.TcDUT
TYPE ST_PACK_CodeBuffer :
STRUCT
	sBuffer			: ARRAY[1..2] OF ST_PACK_CodeStatus;
END_STRUCT
END_TYPE

// ---- DUTs/METS/Packs/ST_PACK_CodeStatus.TcDUT
TYPE ST_PACK_CodeStatus :
STRUCT

	strCode			: T_PACK_Barcode;
	strCodeToHMI		: T_PACK_Barcode;
	aCode			: ARRAY[1..4] OF T_PACK_Barcode;
	nStringSize		: INT;
	nStatus			: BYTE;
	nCameraIndex		: INT;
	nScanNo			: INT;
	fXPos			: LREAL;
	fYPos			: LREAL;
	nProgramNo		: BYTE;
	nTriggerID 		: UDINT;
END_STRUCT
END_TYPE

// ---- DUTs/METS/Packs/ST_PACK_ConfirmationQueue.TcDUT
TYPE ST_PACK_ConfirmationQueue :
STRUCT

	nIndex				: INT;				(* number of Outers in queue *)
	sLastBarcode			: ST_SCANNER_ImageData;	(* last Outer barcode added to Infeed Queue *)
	aPackQueue			: ARRAY[1..10] OF ST_SCANNER_ImageData; (* Infeed queue *)

END_STRUCT
END_TYPE

// ---- DUTs/METS/Packs/ST_PACK_Data.TcDUT
TYPE ST_PACK_Data :
STRUCT
	sPackCode			: T_PACK_Barcode;		(*explicitee Pack barcode in case will be neccesary modified it comapre to scanner data*)
	nPackTriggerID			: UDINT;	(* TriggerID value for scanners *)
	sProductionDate		: STRING(10);
	sProductionTime		: STRING(8);
	sProductionTimeOffset	: STRING(6);		(* time offset between system and UTC, '+1:00' means SystemTime = UTC + 1hr *)
	sPackTimeStamp			: T_ISO8601Time;
	nPackStatus			: BYTE;		(*Match to OACPackStatus*)
	sPackRejectCode		: T_RejectCode;
	nPackRejectID			: UINT;
	(*nPackSUPIResult		: DINT;	(* Pack code SUPI status *)*)
	ePackCodeFilledIn		: E_PACK_FilledInStatus;	(* Pack code filled in by first/secondary master list/removed  *)
	stPackCodeData		: ST_SCANNER_CodeData; (* Infeed queue *)
END_STRUCT
END_TYPE

// ---- DUTs/METS/Packs/ST_PACK_InfeedQueue.TcDUT
TYPE ST_PACK_InfeedQueue :
STRUCT
	nIndex				: INT;				(* number of Outers in queue *)
	(*bDoorReject			: BOOL;*)
	sLastBarcode			: T_PACK_Barcode;	(* last Outer barcode added to Infeed Queue *)
	aPackQueue			: ARRAY[1..cMAX_PACK_INFEED_QUEUE] OF ST_PACK_Data; (* Infeed queue *)

END_STRUCT
END_TYPE

// ---- DUTs/METS/Packs/ST_PACK_InTransferQueue.TcDUT
TYPE ST_PACK_InTransferQueue :
STRUCT

	nIndex				: INT;				(* number of Outers in queue *)
	bDoorReject			: BOOL;
	sLastBarcodeAdded		: T_PACK_Barcode;	(* last Outer barcode added to Infeed Queue *)

	aPackQueue			: ARRAY[1..35] OF ST_PACK_Data; (* Stacker queue *)

END_STRUCT
END_TYPE

// ---- DUTs/METS/Packs/ST_PACK_TriggerOffset.TcDUT
TYPE ST_PACK_TriggerOffset :
STRUCT
	nArmPositionOffset			: DINT;	(*position in mm*)
	nCameraPositionOffset		: DINT;	(*position in mm*)
	nTrigger1PositionOffset		: DINT;	(*position in mm*)
	nTrigger2PositionOffset		: DINT;	(*position in mm*)
	nTrigger3PositionOffset		: DINT;	(*position in mm*)
	nTrigger4PositionOffset		: DINT;	(*position in mm*)
	nTrigger5PositionOffset		: DINT;	(*position in mm*)
	nTrigger6PositionOffset		: DINT;	(*position in mm*)
END_STRUCT
END_TYPE

// ---- DUTs/METS/Packs/_Lab/ST_LAB_OuterData_1.TcDUT
TYPE ST_LAB_OuterData_1 :
STRUCT
	sOuterCode			: T_MaxString;
	nOuterStatus		: INT;
	nOuterRejectID		: UINT;
	
	aPacks 				: ARRAY[1..3] OF ST_LAB_PackData;
END_STRUCT
END_TYPE

// ---- DUTs/METS/Packs/_Lab/ST_LAB_PackData_1.TcDUT
TYPE ST_LAB_PackData_1 :
STRUCT
	sPackCode				: T_MaxString;
	nPackStatus				: INT;
	nPackRejectID			: UINT;
END_STRUCT
END_TYPE

// ---- DUTs/METS/PCM/PCM_Hierarchy/ProductInformation/Product/ST_HierarchyData.TcDUT
//{attribute 'pack_mode' := '8'}
TYPE ST_HierarchyData :
STRUCT

	UnitQty 	: STRING(10);
	GTIN 		: T_CodeGTIN;
	EAN 		: STRING(20);
	BCODE9	: T_CodeBRAND;
END_STRUCT
END_TYPE

// ---- DUTs/METS/PCM/PCM_Hierarchy/ProductInformation/Settings/ST_ToleranceThresholdCS.TcDUT
//{attribute 'pack_mode' := '8'}
TYPE ST_ToleranceThresholdCS :
STRUCT
		GoodReadPercentagePAL		:	STRING(6);
END_STRUCT
END_TYPE

// ---- DUTs/METS/PCM/PCM_Hierarchy/ProductInformation/Settings/ST_ToleranceThresholdOUT.TcDUT
//{attribute 'pack_mode' := '8'}
TYPE ST_ToleranceThresholdOUT :
STRUCT
		GoodReadPercentagePAL		:	STRING(6);
		GoodReadPercentageCS		:	STRING(6);
END_STRUCT
END_TYPE

// ---- DUTs/METS/PCM/ST_PCM_Status.TcDUT
//{attribute 'pack_mode' := '8'}
TYPE ST_PCM_Status :
STRUCT
	bEnabled				: BOOL;			(* TRUE = PCM active on machine *)
	bLoaded					: BOOL;			(* TRUE = PCM data loaded *)
	bValid					: BOOL;			(* TRUE = PCM data valid *)
	bTemplateOK				: BOOL;			(* TRUE = all configured printers have templates loaded OK *)

	sPCMCurrent				: T_PCM_Filename;
	sPCMTemplate			: T_PCM_Filename;

	sFieldName				: STRING(255);	(* name of PCM field where validation failed *)
	sFieldData				: STRING(255);	(* data in PCM field where validation failed *)

	sLastFileName			: T_PCM_Filename;(* name of last PCM file loaded *)
	sLastFileTime			: STRING(19);	(* date/time when last PCM file loaded *)
	stLastPCMTime			: TIMESTRUCT;

	sProductionSite 		: STRING(4);
	sProductionLine			: STRING(4);
	sLocalFactoryProductLine: STRING(4);

	stGS1_AI_Definition		: ST_GS1_AI_Definition;

	bOpModeChanged			: BOOL;			(* TRUE = <CodingAndTrackingMode> has changed *)
	bPackGTINChanged		: BOOL;			(* TRUE = <PACK GTIN> has changed *)
	bOuterGTINChanged		: BOOL;			(* TRUE = <OUTER GTIN> has changed *)
	bCaseGTINChanged		: BOOL;			(* TRUE = <CASE GTIN> has changed *)
	bBatchChanged			: BOOL;			(* TRUE = <BatchID> has changed *)
	bProductionChanged		: BOOL;			(* TRUE = <PrductionOrder> has changed *)
	bRSKUChanged			: BOOL;
	bPitCodeChanged			: BOOL;
	bPackBrandSpecChanged	: BOOL;
	bOuterBrandSpecChanged	: BOOL;
	bCaseBrandSpecChanged	: BOOL;

	sEndMarket				: STRING(10);
	sOuterType				: STRING(5);
	nOpMode					: INT;	(* selected operating mode *)

	sPackGTIN 				: T_CodeGTIN;
	sOuterGTIN 				: T_CodeGTIN;
	sCaseGTIN 				: T_CodeGTIN;

	sBatchNumber			: T_CodeBATCH;
	sProductionOrder		: T_CodePO;
	sRetailSKU 				: T_CodeRSKU;
	sPitCode				: T_CodePIT;

	sPackBrandSpec 			: T_CodeBRAND;
	sOuterBrandSpec 		: T_CodeBRAND;
	sCaseBrandSpec 			: T_CodeBRAND;

	sProductDescription		: T_ProductDescription;

	bEnablePassThrough		: BOOL;			(* enable pass-through mode *)
	bEnableCaseLabels		: BOOL;			(* enable labels on Case *)
	bEnableAggregation		: BOOL;			(* enable aggregation of Outers into Case *)
	bEnableOuterLabels		: BOOL;			(* enable labels on Outer *)
	bEnableOAC				: BOOL;			(* enable old OAC files *)
	bEnableOHM				: BOOL;			(* enable OHM files *)
	bEnablePacks			: BOOL;			(* enable Pack scanners *)

	nAcceptanceLevel		: INT;			(* acceptance level of Packs per Outer for Pack Agregation - In pack numbers NOT %*)

	nCaseAcceptanceLevelPacks	: REAL;			(* acceptance level of Packs per Outer *)
	nOuterAcceptanceLevelPacks	: REAL;			(* acceptance level of Packs per Outer *)
	nCaseAcceptanceLevelOuters	: REAL;			(* acceptance level of Packs per Outer *)

	nPacksPerOuter			: INT;			(* Amount Of  Packs per Outer unit for current PCM *)
	nPacksPerCase			: INT;			(* Amount Of  Packs per Case unit for current PCM *)
	nOutersPerCase			: INT;			(* Amount Of  Outers  per Case unit for current PCM *)

	bReloadPCM				: BOOL;			(* set TRUE to reload local OPI file *)
	(*bBrowsePCM				: BOOL;*)

END_STRUCT
END_TYPE

// ---- DUTs/METS/System/E_SYSTEM_CTState.TcDUT
TYPE E_SYSTEM_CTState :
(
	E_SYSTEMCT_IDLE,
	E_SYSTEMCT_TIMEZONE,
	E_SYSTEMCT_SYSTEMTIME,
	E_SYSTEMCT_SETSYSTEMTIME,
	E_SYSTEMCT_ERROR,
	E_SYSTEMCT_CREATETEMPFOLDER,
	E_SYSTEMCT_CREATEBASEFOLDER,
	E_SYSTEMCT_DONE
);
END_TYPE

// ---- DUTs/METS/System/E_SYSTEM_HandScannerBaudrate.TcDUT
TYPE E_SYSTEM_HandScannerBaudrate :
(
	E_HandScannerBaudrate_IDLE,
	E_HandScannerBaudrate_READ,
	E_HandScannerBaudrate_WRITE,
	E_HandScannerBaudrate_ERROR_READ,
	E_HandScannerBaudrate_ERROR_WRITE,
	E_HandScannerBaudrate_DONE
);
END_TYPE

// ---- DUTs/METS/System/E_SYSTEM_ItemType.TcDUT
TYPE E_SYSTEM_ItemType :
(
	ePack  	:= 0,
	eOuter	:= 1,
	eCase	:= 2,
	eInterim	:= 3
);
END_TYPE

// ---- DUTs/METS/System/E_SYSTEM_MachineState.TcDUT
{attribute 'qualified_only'}
//{attribute 'strict'}
{attribute 'to_string'}
TYPE E_SYSTEM_MachineState :
(
	(*Grey*)
	POWERUP				:=0,

	(*Red*)
	IMMEDIATESTOPPED			:=100,
	MACHINEINERROR			:=110,
	
	(*Yellow*)
	INITIALISING			:=200,
	MANUAL				:=210,

	(*Blue*)
	READYTOSTART		:=300,
	STOPPING						:=310,

	(*Green*)
	RUNNING				:=400,
	WAITINGFORPRODUCT	:=410,
	PASSTHROUGHACTIVE		:=420,
	CONDITIONALRUNNING	:=430
);

END_TYPE

(*
	(*Grey*)
	eSYSTEM_POWER_UP				:=0,

	(*Red*)
	eIMMEDIATE_STOPPED			:=100,
	eMACHINE_IN_ERROR			:=110,

	(*Yellow*)
	eSYSTEM_INITIALISING			:=200,
	eSYSTEM_MANUAL				:=210,

	(*Blue*)
	eSYSTEM_READY_TO_START		:=300,
	eSTOPPING						:=310,

	(*Green*)
	eSYSTEM_RUNNING				:=400,
	eMACHINE_WAITING_FOR_PRODUCT	:=410,
	eCONVEYOR_MODE_ACTIVE		:=420,
	eSYSTEM_CONDITIONAL_RUNNING	:=430
	*)

// ---- DUTs/METS/System/E_SYSTEM_MaintainFolders.TcDUT
TYPE E_SYSTEM_MaintainFolders :
(
	E_FOLDER_IDLE,
	E_FOLDER_ININT_CHECK,
	E_FOLDER_CHECK,
	E_FOLDER_CREATEBASEPATH,
	E_FOLDER_DELETE,
	E_FOLDER_DONE
);
END_TYPE

// ---- DUTs/METS/System/E_SYSTEM_OSType.TcDUT
TYPE E_SYSTEM_OSType : (
	E_OS_UNKNOWN,
	E_OS_WINCE,
	E_OS_WINDOWS
);

END_TYPE

// ---- DUTs/METS/System/Status/ST_SYSTEM_BridgeStatus.TcDUT
//{warning 'CONVERSION MESSAGE: This text contained unprintable characters, that have been deleted'.}
TYPE ST_SYSTEM_BridgeStatus :
STRUCT
	sBridgeVersion				: STRING;
	sFSSServerIpAddress 		: STRING :='10.16.16.27';
	sFSSServerWebRequest	 	: T_MaxString :='Apriso/MessageProcessor/FlexNetMessageProcessor.asmx';
	(*nFSSResponseTimeout		: TIME := t#60s;*)
	nFSSResponseTimeout		: UINT := 60000;
	nBridgeStatus 				: INT; (* Initialized = 0,           (TwincatInitialized = 1,            PLCVariablesInitialized = 2,            ReadProcessVariablesError = 3,            PCMReceiverInitialized = 4,            PCMReceiverRunning = 5,            PCMReceiverNewPCMArrived = 6,            Error = 7,            BridgeInCommissioningMode = 8,            BridgeConnectedToFSS = 9*)
	nBridgeWatchdog 			: INT;
	nBridgeTimeout 			: INT;
	sFaultCodeDirectory 		: STRING :='C:/METS';
	sFSSFaultCodeAge 			: INT :=10;
	sFSSCHMDirectory 			: STRING:='C:/METS/CHM';
	bCommissioningMode		: BOOL;
	bFSSReportsError			: BOOL;
	nFSSResendAttempts 		: INT :=5;

	sLastFileTimeToDlogHMI 		: STRING(255);
	sLastFileNameToDlogHMI 	: STRING(255);

	sDBConnectionString		: STRING(50);
	sLocalBridgePath			: T_FolderPath;
	sLocalCACPath 				: T_FolderPath;

	(*sBridgeUIPath :STRING := 'C:/METS/Bridge/METS_Bridge_UI/METS_Bridge_UI.exe';
	sPLCSymbolsPath :STRING :='C:/METS/Bridge/METS_Bridge_Core/XML/PLC_Variables.xml';
	sADSIp :STRING :='10.185.3.235.1.1';
	sADSPort :STRING :='801';*)
END_STRUCT
END_TYPE

// ---- DUTs/METS/System/Status/ST_SYSTEM_MachineStatus.TcDUT
TYPE ST_SYSTEM_MachineStatus :
STRUCT

	eHWType						: E_CX_HWType;
	eOSType						: E_SYSTEM_OSType;		(* OS type *)
	stHardware					: ST_CxDeviceIdentificationEx;	(* hardware info *)


	bMETSAppOK				: BOOL;
	bMETSLogsOK				: BOOL;	
	bMETSProcessOK			: BOOL;
	bMETSPathsOK			: BOOL;

	
	sMETSAppPath				: T_FolderPath;
	sMETSLogsPath				: T_FolderPath;	
	sMETSProcessPath			: T_FolderPath;
	
	sTCInstalationPath			: T_FolderPath;
	bSystemFoldersOK			: BOOL;
	sFolderStatus				: STRING(25);
	
	sArchiveDBPath			: T_FolderPath;	(*local ArchiveDB path*)
	sBridgeAppPath 			: T_FolderPath;	(* local Bridge path *)
	sLoggerAppPath			: T_FolderPath;	(*  *)
	sWebHMIPath				: T_FolderPath;	(*  *)
	sDeleteArchivePath		: T_FolderPath;	(*  *)
	
	sPCMPath 			: T_FolderPath;	(* local PCM path *)
	sPCMIncomingPath 	: T_FolderPath;	(* local PCM/Incoming path *)
	sCHMPath 			: T_FolderPath;	(* local CHM path *)
	sSettingsPath		 	: T_FolderPath;	(* local Setting*)
	sBackupsPath			: T_FolderPath; (*local Setting/Backup path*)
	sRecipePath				: T_FolderPath; (*local Setting/Recipe path*)
	sCamerasPath				: T_FolderPath;	(* local Camera path *)
	sPrintersPath			: T_FolderPath;	(* local Camera path *)
	
	sOCVPath 			: T_FolderPath;	(* local OCV path *)
	sOACPath 			: T_FolderPath;	(* local OAC path *)
	sCACPath 			: T_FolderPath;	(* local CAC path *)
	sSystemLogPath			: T_FolderPath;	(* local Log path *)
	
	bClearProcessFolders		: BOOL;
	
///////////////////////////////////////////////////////////	
	//bBasePathOK					: BOOL;
	//sBasePath					: T_FolderPath;		(*TO BE REMOVED*)
	//sLocalArchiveDBPath				: T_FolderPath;
	//sLocalBridgePath				: T_FolderPath;
	//sLocalPCMPath 					: T_FolderPath;	(* local PCM path *)
	//sLocalPCMFSSPath 				: T_FolderPath;	(* local PCM/FSS path *)
	//sLocalOCVPath 					: T_FolderPath;	(* local OCV path *)
	//sLocalOACPath 					: T_FolderPath;	(* local OAC path *)
	//sLocalOHMPath 					: T_FolderPath;	(* local OHM path *)
	//sLocalCACPath 					: T_FolderPath;	(* local CAC path *)
	//sLocalCHMPath 					: T_FolderPath;	(* local CHM path *)
	//sLocalKPIPath 					: T_FolderPath;	(* local KPI path *)
	//sLocalHMIPath 					: T_FolderPath;	(* local HMI path *)
	//sLocalSettingsPath 				: T_FolderPath;	(* local Setting path*)
	//sLocalBackupsPath 				: T_FolderPath;	(* local Setting/Backups *)
	//sLocalOrcaPath					: T_FolderPath;	(* local ORCA path *)
	//sLocalSystemLogPath				: T_FolderPath;	(* local SystemLog path *)
////////////////////////////////////////////////////////////////
	bNVDataInitOK				: BOOL;
	bNVDataExport				: BOOL;
	bNVDataImport				: BOOL;

	bMachineConfigReadOK		: BOOL;
	bSettingsValid				: BOOL;
	bSettingsChanged			: BOOL;

	sSettingsErrorField			: STRING(20);
	sSettingsErrorData			: STRING(20);
	nShiftOffsetTime			: DINT;

	bSystemTimeValid			: BOOL;
	stCTDateTime				: ST_SYSTEM_DateTime;
	bNetworkInfoValid			: BOOL;
	stNetworkInfo				: ST_CX_NetworkInfo;

	bTCPServerInitOK			: BOOL;
	bFileDB_OK					: BOOL;		//File mode for ArchiveDB if DB reamin offline
	
	aHMIRunning					: ARRAY[1..2] OF BOOL;
	bArchiveDBRunning			: BOOL;
	bBridgeRunning				: BOOL;
	bLoggerRunning				: BOOL;
	bReportingDBRunning			: BOOL;
	
	bStartUpComplete			: BOOL;			(* All ready! *)

(* *********************************************************** *)
(* ***************        Genreal PLC section	 ************************)
(* *********************************************************** *)

	bReset						: BOOL;		(* must be linked to machine RESET signal *)
	bShortReset					: BOOL;
	bLongReset					: BOOL;
	bHardReset					: BOOL;

	bStartRequest					: BOOL;
	bStopRequest					: BOOL;


	bPowerUpComplete				: BOOL;
	bSystemPowerOK				: BOOL := TRUE;		(* link to external power signal if available *)

	bAllCamerasReadyOK			: BOOL;
	bAllPrintersReadyOK			: BOOL;
	bAllMotorsReadyToRunOK		: BOOL;
	(*bAllCylindersEnableOK			: BOOL;*)
	bAllExternalDeviceOK			: BOOL;
	bAllSeqStationHomed			: BOOL;
	bAllStationNotMoving			: BOOL;
	bPCMReceiverRunning			: BOOL;
	bMETSConnectedToFSS			: BOOL;
	bMETSConectedToDB			: BOOL;
	bMachineReadyToStart			: BOOL;

	stMachineMode				: ST_SYSTEM_MachineMode;
	bMachineEnabled				: BOOL;
	bTPDConditionalEnabled		: BOOL;
	bExternalConditionalEnabled	: BOOL;
	bEUCAConditionalEnabled		: BOOL;

	bMachineRunning				: BOOL;
	bMachineConditionalRunning		: BOOL;
	bMachineWaitingOnProduct		: BOOL;
	bMachineStopped				: BOOL;
	bInternalStopRequest			: BOOL;
	bMachineConveyorMode			: BOOL;

	bUseOverlayPanel					: BOOL;
	bUseLinearPackCodeScreen		: BOOL;
	bUseInterimCodeForValidation	: BOOL;

	nClearQueuesDone				: BYTE;

	bEndOfShift					: BOOL;
	stLastShift						: TIMESTRUCT;

	bEndOfProdOrder				: BOOL;
	stLastProdOrder				: TIMESTRUCT;

	stPCMData					: ST_PCM_Data;
	stPCMStatus					: ST_PCM_Status;

END_STRUCT
END_TYPE

// ---- DUTs/METS/System/Status/ST_SYSTEM_ReportingDBStatus.TcDUT
//{warning 'CONVERSION MESSAGE: This text contained unprintable characters, that have been deleted'.}
TYPE ST_SYSTEM_ReportingDBStatus :
STRUCT
	sReportingDBVersion			: STRING;
	nReportingDBStatus 			: INT;
	nReportingDBWatchdog 		: DINT;
	bReportingDBHealthy			: BOOL;
	
	sPLCVersionHMI				: STRING;
	sPLCVersionInfoHMI			: T_MaxString;

	stMachineID				: ST_SYSTEM_MachineID;
	stMachineState			: ST_SYSTEM_MachineState;
	
	bMainItemReset			: BOOL;
	sStartDateTime			: T_ISO8601Time;		(* last PLC restart*)
	
	nShiftID				: INT;
	
	nCodingAndTrackingMode	: INT;
	sBatchNumber			: T_CodeBATCH;
	sProductionOrder		: T_CodePO;
	sRetailSKU 				: T_CodeRSKU;
	sProductDescription		: T_ProductDescription;
	
	nPacksPerOuter			: INT;			(* Amount Of  Packs per Outer unit for current PCM *)
	nPacksPerCase			: INT;			(* Amount Of  Packs per Case unit for current PCM *)
	nOutersPerCase			: INT;			(* Amount Of  Outers  per Case unit for current PCM *)
	
	aCameraName				: ARRAY[1..cMAX_CAMERA_NUMBER] OF STRING(30);
END_STRUCT
END_TYPE

// ---- DUTs/METS/System/ST_SYSTEM_Config.TcDUT
{attribute 'pack_mode' := '1'}
TYPE ST_SYSTEM_Config :
STRUCT
(*******************************************************************************************************************************************************)
(*********************************************************General EUCA-TPD*******************************************************************************)
(*******************************************************************************************************************************************************)
(*General screen*)
	sBackupName								: STRING;
	sProductionSite 							: STRING(4);
	stProductionLine 							: ST_SYSTEM_ProductionLine;
	sShiftOffsetTime							: STRING(6);	(* shift offset time, formatted as '-06:00' or '+02:00' *)
	stSoftVersion								: ST_SYSTEM_SoftwareVersion;

	sFC1ReplacmentChar						: STRING(1) := '';

(*FSS settings*)
	tFSSLostConnectionTimeOut				: TIME := t#30m;
	sFSS_Server_IPAddress						: STRING:= '127.0.0.1'; (*Do not remove. Used for HMI*)
	sFSS_Server_WebRequest					: T_MaxString := 'http://127.0.0.1/Apriso/MessageProcessor/FlexNetMessageProcessor.asmx'; (*Do not removed. Used for HMI - this is the CHM sending endpoint*)
	nFSSResponseTimeout						: UINT := 60000; (*: TIME := t#60s;*)
	nFSSResendAttempts						: INT := 5;

(*Shift Setup schedule*)
	aShiftSchedule								: ARRAY[1..cSHIFTNUMBER] OF TIMESTRUCT;
	aShiftChangeActive							: ARRAY[1..cSHIFTNUMBER] OF BOOL;

(*Door*)
	stDoorSettingsZone1					: ST_SYSTEM_Door;
	stDoorSettingsZone2					: ST_SYSTEM_Door;

(*Barcode setup - NEW - Gradually implementing*)
	stCodeInfo_Pack								: ST_CodeInfo :=		(eCodeType :=E_PACK);
	stCodeInfo_Intermediate						: ST_CodeInfo :=		(eCodeType :=E_INTERIM);
	stCodeInfo_Outer								: ST_CodeInfo :=		(eCodeType :=E_OUTER);
	stCodeInfo_Case								: ST_CodeInfo :=		(eCodeType :=E_CASE);

(*******************************************************************************************************************************************************)
(********************************************************Switch******************************************************************************)
(*******************************************************************************************************************************************************)
(*General Switches*)
	bEUCAMonitor24VSupply					: BOOL := TRUE;
	bMonitorRemote24VSupply				: BOOL;
	bInhibitSafetyResetWhenAirNOK			: BOOL;

	bKPIRemoteShareEnable					: BOOL;
	bSystemLogEnable							: BOOL := TRUE;
	bArchiveDBEnable							: BOOL := TRUE;
	bPassthrough								: BOOL;
	bPassthroughTPD							: BOOL;
	bHandScannerInMainCabinet				: BOOL; (**)
	bValidateOCVOnly							: BOOL;
	bEnableRestoreOCV						: BOOL;		(*Enable Restoring of OCV data from structure*)
	bATTPModeEnable							: BOOL := TRUE;

	bConditionalStateAllowed					: BOOL := TRUE;
	bNoStationsAvailable						: BOOL := TRUE;
	bCommisioningMode						: BOOL; 	(**)
	bConveyorAsPreMachine					: BOOL := TRUE;

	bExistPreTPDBuildBackSensor				: BOOL := TRUE;
	bExistTPDExitBlockedSensor				: BOOL := TRUE;
	bExistPreEUCABuildBackSensor			: BOOL;
	bExistEUCAExitBlockedSensor				: BOOL;
	bExistWrapperPackRejectSesnor			: BOOL;

(*Enable Master List Fillin*)
	bEnablePackPrimaryMasterList					: BOOL:=TRUE;
	bEnablePackSecondaryMasterList				: BOOL:=TRUE;
	bEnableOuterMasterList						: BOOL:=TRUE;

	bExtendedDiagnosticEnable				: BOOL;
	bDotCodeFormat								: BOOL;
	bQRCodeFormat								: BOOL;

(*Pack*)
	bEnableFastArming							: BOOL:=TRUE;		(*Enable arming sensors even if outer did not leave Lightox yet *)
	bPAOLIsolatorExist						: BOOL;
	bLightbox4TrigerSystemExist				: BOOL;
	bLightboxLensAirExist						: BOOL;
	bLighboxOverCMLConveyor					: BOOL;
	bLightboxCamerasOnFullResolution				: BOOL;
	bCloseCameraRelay						: BOOL;
	bPackSeparatorAnalogControl				: BOOL;
	bCameraOnLeftSide							: BOOL; 	(*Set to true if the camera is on the left hand side of the conveyor as the packs travel trhough it towards the CML*)
	bPackCodesTrailing							: BOOL := TRUE; 	(*Set to true if the pack codes are on the trailing edge of the pack as it travels through the infeed cameras*)
	bFirstPackCodeOnTop							: BOOL;			(*Used for correct mapping packs from pack confirmation camera*)

	bEnableCodeAdjustment						: BOOL;
	bEnableCodeDuplicateCheck					: BOOL;
	bExtendedOCVDupCheck						: BOOL;
	bLinearPackBufferExist							: BOOL;
	bEnableStopForInvalideCode					: BOOL;	(*Stop METS immidiatly after Lightbox detect invalide code*)
	bEnablePackCodeDateCheck					: BOOL;
	bFixedTriggerOffsetEnable						: BOOL;

(*Outer*)
	bFrontConfirmationCameraInUse			: BOOL;				(*Rear confirmation camera 192.168.1.41 = false, front confiramtion camera 192.168.1.42 = true*)
	bEnableOuterRejectConfirmation			: BOOL;
	bEnableOuterTransferConfirmation		: BOOL;
	bMasterListCameraDoubleRead				: BOOL := TRUE;
	bAggregationCameraRunWithTrigger			: BOOL;
	bAggregationStopOnInvalidCode				: BOOL ;
	bUseAuxRowCompleteSesnor					: BOOL;
	bUseInterimCodeForLastPosition				: BOOL;
	bSkipStopGate									: BOOL;
	bPreLabelerShiftRegUsed						: BOOL;
	bConfirmOnOuter								: BOOL;		(*At Focke NCW outer is confirmet by it last packs*)
	bEanbleRestoreOCVFromConfirmation			: BOOL;		(*At Focke NCW two outers will be resotred after index = 2 x pack per outers*)
	bExtendedOACDupCheck						: BOOL;

(*Case*)
	bPushIntoCaseCount							: BOOL;
	bIntermediateBufferExist						: BOOL;
	bCasePackerDirectCutOut						: BOOL;
	bCasePositionOverwritingCheck				: BOOL := TRUE;
	bAddOACFromFileOnly						: BOOL;	(*Add OAC to infeed from file not from arrOuterStatus*)
	bSentOnlyGoodHierarchy						: BOOL := TRUE;
	bArchiveRejectedHierarchy					: BOOL := TRUE;
	bEnableStopOnOverWrittenData				: BOOL;
	bResetPushCountOnDoorOpen				: BOOL;
	bCheckDuplicateCaseLabel					: BOOL;
	bManualConfirmationEnable					: BOOL;
	bEnableStopOnCaseInavlid						: BOOL;
	bUseCaseFullAsValidationTrigger				: BOOL;
	bUseCaseContentReject						: BOOL;
	bUseRejectByCasepacker						: BOOL;
	bAggregationWithoutCamera					: BOOL;
	bOrcaExist										: BOOL;

(*Commisioning settings*)
	bDisableOuterReject						: BOOL;	(*Disable any outer reject - just for commisioning*)
	bDisableCaseReject						: BOOL;	(*Disable any case reject - just for commisioning*)
	bOuterRejectWithHighSignal				: BOOL;
	bCaseRejectWithHighSignal				: BOOL;

(* Device Settings*)
	bUPSExist										: BOOL;
	bUPSImmediateShutdown						: BOOL := FALSE;		(*Option to control immediate shutdown on power loss*)

	bApplyLabelInPassthrough					: BOOL;
	bDisableApplyLabel						: BOOL;
	bPrinterHighSpeedEnable					: BOOL;
	bEANValidationEnable						: BOOL;

	bPrintSignalFromPLC						: BOOL;
	bEnableResendCommand					: BOOL;

(*******************************************************************************************************************************************************)
(********************************************************Numercis******************************************************************************)
(*******************************************************************************************************************************************************)
(*Line system type set up*)
	nPackAggregationMode						: INT := 0; (* 0 -NOPACKAGGREGATION, 1 -STRUCTURALAGGREGATION (PAOL), 2 -STRUCTURALAGGREGATION (2CAM),  3 - LINEARAGGREGATION (PLAS), 4 - NCWAGGREGATION (PLAS + INTERIM)*)
	nOuterAggregationMode						: INT := 0; (* 0 - SYNCHROCONFIRMATION, 1 - SHIFTCONFIRMATION, 2 -SFLXNOCONFIRMATION, 3 - SFLXWITHCONFIRMATION, 4 - LASERPRINTLABEL*)
	nAutomationMode								: INT := 0; (* 0 - EXTERNAL, 1 - CML, 2 - LARS, 3 - SIDEFLEX *)

(* Consecutive rejects counter*)
	nConsecutivePackRejects						: UINT := 3;
	nConsecutivePackConfirmationMissing		: UINT := 3;
	nConsecutiveOCVMissing						: UINT := 3;
	nConsecutiveIntermediateNoRead				: UINT := 3;
	nConsecutiveOuterRejects						: UINT := 3;
	nConsecutiveCaseContentMissing				: UINT := 3;
	nConsecutiveCaseRejects						: UINT := 3;

(*Archive settings*)
	nMaximumArchiveAge							: INT := 28;		(*Max archive age in days*)
	nMaximumArchiveFiles						: INT := 100;

	nMaximumOCVFiles							: INT := 5000;
	nMaximumOACFiles							: INT := 1000;
	nMaximumErrorFiles							: INT := 100;

(* HMI settings*)
	nWarningLevelPack							: REAL := 99.95;
	nAlarmLevelPack								: REAL := 99.9;
	nWarningLevelOuter							: REAL := 99.5;
	nAlarmLevelOuter								: REAL := 99.0;
	nWarningLevelCase							: REAL := 99.5;
	nAlarmLevelCase								: REAL := 95.0;

	tPassthroughDisableDelay						: TIME := t#2s;
(*SequenceTimeOut*)
	tPackMasterListTimeout						: TIME := t#250ms;
	tPackAgreggationTimeout						: TIME := t#500ms;
	tPackConfirmationTimeout					: TIME := t#500ms;
	tInterimTimeout								: TIME := T#500ms;
	tOuterValidationTimeout						: TIME := t#750ms;
(*Sensors Timeouts*)
	tRejectSensorTimeout							: TIME := T#10s;
	tRowCompleteSignalTimeOut					: TIME := t#25s;
	tLayerCompleteSignalTimeOut					: TIME := t#25s;
	tIntermediatePushSignalTimeOut				: TIME := t#25s;
	tCaseCompleteSignalTimeOut					: TIME := t#25s;
	tDischargeSignalTimeOut						: TIME := t#25s;
	tCaseLabelValidationSignalTimeOut			: TIME := t#25s;
	tCaseRejectTimeOut							: TIME := t#60s;

(*Pack*)
	nAggregationUnitLightingIntensityTop		: INT := 100;		(*to be removed and replaced with camera config*)
	nAggregationUnitLightingIntensity			: INT := 100;				(*to be removed and replaced with camera config*)
	tLightboxLensAirFrequency					: TIME := t#3h;
	tLightboxLensAirBlowDuration				: TIME := t#10s;
	nClearPMLIndex								: INT;
	nClearPMLRecords								: INT;
	stPackAgregationCameraOffset				: ST_PACK_TriggerOffset;	(*Used for SFLX 2 Cam aggregation*)
	stPackCamera01Offset							: ST_PACK_TriggerOffset;	(*Used for SFLX 2 Cam aggregation*)
	stPackCamera02Offset							: ST_PACK_TriggerOffset;	(*Used for SFLX 2 Cam aggregation*)

	nConfirmationPackCode1						: INT := 1;
	nConfirmationPackCode2						: INT := 2;
	nPacksPerStack								: UINT := 5;
	nMaxOutersBuffer								: UINT := 1; 		(*Maximum number of outers that can be processes at one time allowing for camera buffers - can be set higher if camera sequence max buffer is fixed!*)
	tBufferDelayTime								: TIME := t#200ms; 		(*Adjust this time so each outer stops for a moment before the first infeed camera sensor in order to avoid out of sync errors*)
	nCheckStatusOCV								: BYTE := 2;
	nExpectedValidationDepth						: INT := 1;
	nInterimQueueIndex							: INT :=1;

(*Outer*)
	nOutersPerRow									: INT := 5;
	tTwoOutersOnRejectConv						: TIME := T#500ms;
	nMasterListNumbersWarning					: INT := 5;
	nAuxRowCount								: INT := 2;
	nAggregationQueueIndex						: INT := 0;
	tInspectionDelay								: TIME := t#30ms;

(* Case*)
	nCaseQueueLength							: INT := 3;
	nCaseContentBuffer							: INT;

(*Device*)
	tUPSShutdownDelay							: TIME := t#30s;		(*Default grace period for NT_Shutdown FB*)

(*******************************************************************************************************************************************************)
(********************************************************Devices******************************************************************************)
(*******************************************************************************************************************************************************)
(*Camera - IP/Port settings for All scanners used in EUCA-TPD  arrays with up to 6 scanners per array *)
	aCameraSettings							: ARRAY [1..cMAX_CAMERA_NUMBER] OF ST_SCANNER_Config;

(*Printers*)
	aPrinterSettings							: ARRAY [1..cMAX_PRINTER_NUMBER] OF ST_PRINTER_Config;

(*Hand Scanners*)
	aHandScannersConfig						: ARRAY [1..cMAX_HAND_SCANNERS] OF ST_SCANNER_HoneywellConfig;
	aHoneywellCtrl								: ARRAY [1..cMAX_HAND_SCANNERS] OF ST_SCANNER_HoneywellCtrl;
	stUSBScannerConfig						: ST_SCANNER_USBConfig;

(* Profinet drives *)
	aProfiNetMaster							: ARRAY [1..cMAX_PROFINET_MASTERS]  OF  ST_ProfinetMasterConfig; (* EL6631 *)
	aProfiNetDrive								: ARRAY [1..cMAX_PROFINET_DRIVES]  OF ST_ProfinetDrive; (*config for individual drives *)

(*MC2 drives*)
	aAxisConfig								: ARRAY [1..cMAX_MC2_DRIVES] OF ST_AXIS_Config;

(* Analog drive*)
	stPackSeparator							: ST_AnalogDrive;

(*Cylinders*)
	aCylinderConfig							: ARRAY [1..cMAX_CYLINDERS] OF ST_CYLINDER_Config;

(* CAMS  *)
	(*aAFS50camConfig						: ARRAY [1.. cMAX_CAMS] OF ST_AFS60_Config;*)

(*Database*)
	(*stDBConfig								: ST_DB_Config;*)

(*******************************************************************************************************************************************************)
(********************************************************Single IO******************************************************************************)
(*******************************************************************************************************************************************************)
(*Single Input Config*)
	st_I_TransferCoveyorDoorGuard1			: ST_IO2_SingleInputCtrl:=			(eTypeInput:=E_IO2_Type.NO,		tTimeOnFilter:=t#100ms, 		tTimeOffFilter:=t#10ms, 	sInputName:='Transfer Coveyor Door Guard 1' );	(**)
	st_I_TransferCoveyorDoorGuard2			: ST_IO2_SingleInputCtrl:=			(eTypeInput:=E_IO2_Type.NO,		tTimeOnFilter:=t#100ms, 		tTimeOffFilter:=t#10ms, 	sInputName:='Transfer Coveyor Door Guard 2' );	(**)

	st_I_DoorOpenZone1					: ST_IO2_SingleInputCtrl:=			(eTypeInput:=E_IO2_Type.NO,		tTimeOnFilter:=t#100ms, 		tTimeOffFilter:=t#10ms, 	sInputName:='Door Open Zone 1' );	(**)
	st_I_DoorOpenZone2					: ST_IO2_SingleInputCtrl:=			(eTypeInput:=E_IO2_Type.NO,		tTimeOnFilter:=t#100ms, 		tTimeOffFilter:=t#10ms, 	sInputName:='Door Open Zone 2' );	(**)

	st_I_AuxRowCompleteSesnor			: ST_IO2_SingleInputCtrl:=			(eTypeInput:=E_IO2_Type.NO,		tTimeOnFilter:=t#10ms, 		tTimeOffFilter:=t#10ms, 	sInputName:='Aux Row Complete' );	(**)
	st_I_CaseRejectedByCasePacker		: ST_IO2_SingleInputCtrl:=			(eTypeInput:=E_IO2_Type.NO,		tTimeOnFilter:=t#10ms, 		tTimeOffFilter:=t#10ms, 	sInputName:='Case Rejected By Casepacker' );	(**)

	st_I_PreMachineAutoRun				: ST_IO2_SingleInputCtrl:=			(eTypeInput:=E_IO2_Type.NO,		tTimeOnFilter:=t#100ms, 		tTimeOffFilter:=t#0ms, 	sInputName:='PreMachine AutoRun' );	(**)
	st_I_CasePackerAutoRun				: ST_IO2_SingleInputCtrl:=			(eTypeInput:=E_IO2_Type.NO,		tTimeOnFilter:=t#100ms, 		tTimeOffFilter:=t#0ms, 	sInputName:='Casepacker AutoRun' );	(**)

	st_I_QAButtonRejectOuter				: ST_IO2_SingleInputCtrl:=			(eTypeInput:=E_IO2_Type.NO,		tTimeOnFilter:=t#100ms, 		tTimeOffFilter:=t#0ms, 	sInputName:='QA Button Reject Outer' );	(**)
	st_I_OuterAtRejectStation				: ST_IO2_SingleInputCtrl:=			(eTypeInput:=E_IO2_Type.NO,		tTimeOnFilter:=t#1000ms, 		tTimeOffFilter:=t#0ms, 	sInputName:='Outer At Reject Station' );	(**)
	st_I_OuterRejectConfirm				: ST_IO2_SingleInputCtrl:=			(eTypeInput:=E_IO2_Type.NO,		tTimeOnFilter:=t#1000ms, 		tTimeOffFilter:=t#0ms, 	sInputName:='Outer Reject Confirm' );	(**)
	st_I_RejectBinFull						: ST_IO2_SingleInputCtrl:=			(eTypeInput:=E_IO2_Type.NO,		tTimeOnFilter:=t#100ms, 		tTimeOffFilter:=t#0ms, 	sInputName:='Reject Bin Full' );	(**)

	st_I_EUCABuildBackPreMachine			: ST_IO2_SingleInputCtrl:=			(eTypeInput:=E_IO2_Type.NO,		tTimeOnFilter:=t#1000ms, 		tTimeOffFilter:=t#0ms, 	sInputName:='EUCA Buildback Sensor' );	(**)
	st_I_EUCAExitBlocked						: ST_IO2_SingleInputCtrl:=			(eTypeInput:=E_IO2_Type.NO,		tTimeOnFilter:=t#1000ms, 		tTimeOffFilter:=t#0ms, 	sInputName:='EUCA Exit Blocked Sensor' );	(**)

	st_I_OuterAtSystemInfeed					: ST_IO2_SingleInputCtrl:=			(eTypeInput:=E_IO2_Type.NO,		tTimeOnFilter:=t#1000ms, 		tTimeOffFilter:=t#0ms, 	sInputName:='Outer At System Infeed Sensor' );	(**)
	st_I_OuterAtAdditionalConv				: ST_IO2_SingleInputCtrl:=			(eTypeInput:=E_IO2_Type.NO,		tTimeOnFilter:=t#1000ms, 		tTimeOffFilter:=t#0ms, 	sInputName:='Outer At Additional Conv Sensor' );	(**)

	st_I_TransferConveyorPlugConnected		: ST_IO2_SingleInputCtrl:=			(eTypeInput:=E_IO2_Type.NO,		tTimeOnFilter:=t#100ms, 		tTimeOffFilter:=t#100ms, 	sInputName:='Transfer Conveyor Plug Connected' );	(**)
	st_I_OutfeedConveyorPlugConnected		: ST_IO2_SingleInputCtrl:=			(eTypeInput:=E_IO2_Type.NO,		tTimeOnFilter:=t#100ms, 		tTimeOffFilter:=t#100ms, 	sInputName:='Outfeed Conveyor Plug Connected' );	(**)
	st_I_AdditionalConveyorPlugConnected	: ST_IO2_SingleInputCtrl:=			(eTypeInput:=E_IO2_Type.NO,		tTimeOnFilter:=t#100ms, 		tTimeOffFilter:=t#100ms, 	sInputName:='Outfeed Conveyor Plug Connected' );	(**)

(*Single Input Config for camera triggers*)
	st_I_Camera01						: ST_IO2_SingleInputCtrl:=			(eTypeInput:=E_IO2_Type.NO,		tTimeOnFilter:=t#6ms, 		tTimeOffFilter:=t#20ms, 	sInputName:='Camera 01' );	(**)
	st_I_Camera02						: ST_IO2_SingleInputCtrl:=			(eTypeInput:=E_IO2_Type.NO,		tTimeOnFilter:=t#6ms, 		tTimeOffFilter:=t#20ms, 	sInputName:='Camera 02' );	(**)
	st_I_Camera03						: ST_IO2_SingleInputCtrl:=			(eTypeInput:=E_IO2_Type.NO,		tTimeOnFilter:=t#6ms, 		tTimeOffFilter:=t#20ms, 	sInputName:='Camera 03' );	(**)
	st_I_Camera04						: ST_IO2_SingleInputCtrl:=			(eTypeInput:=E_IO2_Type.NO,		tTimeOnFilter:=t#10ms, 		tTimeOffFilter:=t#0ms, 	sInputName:='Camera 04' );	(**)
	st_I_Camera05						: ST_IO2_SingleInputCtrl:=			(eTypeInput:=E_IO2_Type.NO,		tTimeOnFilter:=t#10ms, 		tTimeOffFilter:=t#0ms, 	sInputName:='Camera 05' );	(**)
	st_I_Camera06						: ST_IO2_SingleInputCtrl:=			(eTypeInput:=E_IO2_Type.NO,		tTimeOnFilter:=t#10ms, 		tTimeOffFilter:=t#0ms, 	sInputName:='Camera 06' );	(**)
	st_I_Camera07						: ST_IO2_SingleInputCtrl:=			(eTypeInput:=E_IO2_Type.NO,		tTimeOnFilter:=t#10ms, 		tTimeOffFilter:=t#0ms, 	sInputName:='Camera 07' );	(**)
	st_I_Camera08						: ST_IO2_SingleInputCtrl:=			(eTypeInput:=E_IO2_Type.NO,		tTimeOnFilter:=t#10ms, 		tTimeOffFilter:=t#0ms, 	sInputName:='Camera 08' );	(**)
	st_I_Camera09						: ST_IO2_SingleInputCtrl:=			(eTypeInput:=E_IO2_Type.NO,		tTimeOnFilter:=t#10ms, 		tTimeOffFilter:=t#0ms, 	sInputName:='Camera 09' );	(**)
	st_I_Camera10						: ST_IO2_SingleInputCtrl:=			(eTypeInput:=E_IO2_Type.NO,		tTimeOnFilter:=t#10ms, 		tTimeOffFilter:=t#0ms, 	sInputName:='Camera 10' );	(**)
	st_I_Camera11						: ST_IO2_SingleInputCtrl:=			(eTypeInput:=E_IO2_Type.NO,		tTimeOnFilter:=t#10ms, 		tTimeOffFilter:=t#0ms, 	sInputName:='Camera 11' );	(**)
	st_I_Camera12						: ST_IO2_SingleInputCtrl:=			(eTypeInput:=E_IO2_Type.NO,		tTimeOnFilter:=t#10ms, 		tTimeOffFilter:=t#0ms, 	sInputName:='Camera 12' );	(**)

(*METS Cylinders Filtered Inputs *)
	st_I_ClampCylinderExtended		: ST_IO2_SingleInputCtrl:=			(eTypeInput:=E_IO2_Type.NO,		tTimeOnFilter:=t#10ms, 		tTimeOffFilter:=t#0ms, 	sInputName:='Clamp Cylinder Extended' );	(**)
	st_I_ClampCylinderRetracted		: ST_IO2_SingleInputCtrl:=			(eTypeInput:=E_IO2_Type.NO,		tTimeOnFilter:=t#10ms, 		tTimeOffFilter:=t#0ms, 	sInputName:='Clamp Cylinder Retracted' );	(**)

	st_I_GateCylinderExtended		: ST_IO2_SingleInputCtrl:=			(eTypeInput:=E_IO2_Type.NO,		tTimeOnFilter:=t#10ms, 		tTimeOffFilter:=t#0ms, 	sInputName:='Gate Cylinder Extended' );	(**)
	st_I_GateCylinderRetracted 		: ST_IO2_SingleInputCtrl:=			(eTypeInput:=E_IO2_Type.NO,		tTimeOnFilter:=t#10ms, 		tTimeOffFilter:=t#0ms, 	sInputName:='Gate Cylinder Retracted' );	(**)

	st_I_RejectCylinderExtended		: ST_IO2_SingleInputCtrl:=			(eTypeInput:=E_IO2_Type.NO,		tTimeOnFilter:=t#10ms, 		tTimeOffFilter:=t#0ms, 	sInputName:='Reject Cylinder Extended' );	(**)
	st_I_RejectCylinderRetracted 		: ST_IO2_SingleInputCtrl:=			(eTypeInput:=E_IO2_Type.NO,		tTimeOnFilter:=t#10ms, 		tTimeOffFilter:=t#0ms, 	sInputName:='Reject Cylinder Retracted' );	(**)

	st_I_AdditionalRejectCylinderExtended		: ST_IO2_SingleInputCtrl:=			(eTypeInput:=E_IO2_Type.NO,		tTimeOnFilter:=t#10ms, 		tTimeOffFilter:=t#0ms, 	sInputName:='Reject Cylinder Extended' );	(**)
	st_I_AdditionalRejectCylinderRetracted 		: ST_IO2_SingleInputCtrl:=			(eTypeInput:=E_IO2_Type.NO,		tTimeOnFilter:=t#10ms, 		tTimeOffFilter:=t#0ms, 	sInputName:='Reject Cylinder Retracted' );	(**)

	st_I_FirstPusherCylinderExtended		: ST_IO2_SingleInputCtrl:=			(eTypeInput:=E_IO2_Type.NO,		tTimeOnFilter:=t#10ms, 		tTimeOffFilter:=t#0ms, 	sInputName:='Reject Cylinder Extended' );	(**)
	st_I_FirstPusherCylinderRetracted 		: ST_IO2_SingleInputCtrl:=			(eTypeInput:=E_IO2_Type.NO,		tTimeOnFilter:=t#10ms, 		tTimeOffFilter:=t#0ms, 	sInputName:='Reject Cylinder Retracted' );	(**)

	st_I_SecondPusherCylinderExtended		: ST_IO2_SingleInputCtrl:=			(eTypeInput:=E_IO2_Type.NO,		tTimeOnFilter:=t#10ms, 		tTimeOffFilter:=t#0ms, 	sInputName:='Reject Cylinder Extended' );	(**)
	st_I_SecondPusherCylinderRetracted 		: ST_IO2_SingleInputCtrl:=			(eTypeInput:=E_IO2_Type.NO,		tTimeOnFilter:=t#10ms, 		tTimeOffFilter:=t#0ms, 	sInputName:='Reject Cylinder Retracted' );	(**)

(*METS Labellers Filtered Inputs *)
	st_I_Labeller1InPosition					: ST_IO2_SingleInputCtrl:=			(eTypeInput:=E_IO2_Type.NO,		tTimeOnFilter:=t#10ms, 		tTimeOffFilter:=t#0ms, 	sInputName:='Labeller1 In Position' );	(**)
	st_I_Labeller1OuterAtLabeller				: ST_IO2_SingleInputCtrl:=			(eTypeInput:=E_IO2_Type.NO,		tTimeOnFilter:=t#10ms, 		tTimeOffFilter:=t#0ms, 	sInputName:='Labeller1 Outer At Labeller' );	(**)
	tLabeller1OuterAtLabellerTimeLatch		: TIME := t#200ms; (*Variable used separately to keep one standard with HMI user controls for Single Inputs*)

	st_I_Labeller1Ready						: ST_IO2_SingleInputCtrl:=			(eTypeInput:=E_IO2_Type.NO,		tTimeOnFilter:=t#10ms, 		tTimeOffFilter:=t#0ms, 	sInputName:='Labeller1 Ready' );	(**)
	st_I_Labeller1DataReady					: ST_IO2_SingleInputCtrl:=			(eTypeInput:=E_IO2_Type.NO,		tTimeOnFilter:=t#10ms, 		tTimeOffFilter:=t#0ms, 	sInputName:='Labeller1 Data Ready' );	(**)
	st_I_Labeller1HomePosition				: ST_IO2_SingleInputCtrl:=			(eTypeInput:=E_IO2_Type.NO,		tTimeOnFilter:=t#10ms, 		tTimeOffFilter:=t#0ms, 	sInputName:='Labeller1 Home Position' );	(**)
	st_I_Labeller1LabelPrinted					: ST_IO2_SingleInputCtrl:=			(eTypeInput:=E_IO2_Type.NO,		tTimeOnFilter:=t#10ms, 		tTimeOffFilter:=t#0ms, 	sInputName:='Labeller1 Label Printed' );	(**)
	st_I_Labeller1ReadyToApply				: ST_IO2_SingleInputCtrl:=			(eTypeInput:=E_IO2_Type.NO,		tTimeOnFilter:=t#10ms, 		tTimeOffFilter:=t#0ms, 	sInputName:='Labeller1 Ready To Apply' );	(**)
	st_I_Labeller1ApplyDone					: ST_IO2_SingleInputCtrl:=			(eTypeInput:=E_IO2_Type.NO,		tTimeOnFilter:=t#10ms, 		tTimeOffFilter:=t#0ms, 	sInputName:='Labeller1 Apply Done' );	(**)
	st_I_Labeller1SummaryWarning			: ST_IO2_SingleInputCtrl:=			(eTypeInput:=E_IO2_Type.NO,		tTimeOnFilter:=t#10ms, 		tTimeOffFilter:=t#0ms, 	sInputName:='Labeller1 Summary Warning' );	(**)
	st_I_Labeller1Error							: ST_IO2_SingleInputCtrl:=			(eTypeInput:=E_IO2_Type.NO,		tTimeOnFilter:=t#10ms, 		tTimeOffFilter:=t#0ms, 	sInputName:='Labeller1 Error' );	(**)


	st_I_Labeller2InPosition					: ST_IO2_SingleInputCtrl:=			(eTypeInput:=E_IO2_Type.NO,		tTimeOnFilter:=t#10ms, 		tTimeOffFilter:=t#0ms, 	sInputName:='Labeller2 In Position' );	(**)
	st_I_Labeller2OuterAtLabeller				: ST_IO2_SingleInputCtrl:=			(eTypeInput:=E_IO2_Type.NO,		tTimeOnFilter:=t#10ms, 		tTimeOffFilter:=t#0ms, 	sInputName:='Labeller2 Outer At Labeller' );	(**)
	tLabeller2OuterAtLabellerTimeLatch		: TIME := t#40ms; (*Variable used separately to keep one standard with HMI user controls for Single Inputs*)

	st_I_Labeller2Ready						: ST_IO2_SingleInputCtrl:=			(eTypeInput:=E_IO2_Type.NO,		tTimeOnFilter:=t#10ms, 		tTimeOffFilter:=t#0ms, 	sInputName:='Labeller2 Ready' );	(**)
	st_I_Labeller2DataReady					: ST_IO2_SingleInputCtrl:=			(eTypeInput:=E_IO2_Type.NO,		tTimeOnFilter:=t#10ms, 		tTimeOffFilter:=t#0ms, 	sInputName:='Labeller2 Data Ready' );	(**)
	st_I_Labeller2HomePosition				: ST_IO2_SingleInputCtrl:=			(eTypeInput:=E_IO2_Type.NO,		tTimeOnFilter:=t#10ms, 		tTimeOffFilter:=t#0ms, 	sInputName:='Labeller2 Home Position' );	(**)
	st_I_Labeller2LabelPrinted					: ST_IO2_SingleInputCtrl:=			(eTypeInput:=E_IO2_Type.NO,		tTimeOnFilter:=t#10ms, 		tTimeOffFilter:=t#0ms, 	sInputName:='Labeller2 Label Printed' );	(**)
	st_I_Labeller2ReadyToApply				: ST_IO2_SingleInputCtrl:=			(eTypeInput:=E_IO2_Type.NO,		tTimeOnFilter:=t#10ms, 		tTimeOffFilter:=t#0ms, 	sInputName:='Labeller2 Ready To Apply' );	(**)
	st_I_Labeller2ApplyDone					: ST_IO2_SingleInputCtrl:=			(eTypeInput:=E_IO2_Type.NO,		tTimeOnFilter:=t#10ms, 		tTimeOffFilter:=t#0ms, 	sInputName:='Labeller2 Apply Done' );	(**)
	st_I_Labeller2SummaryWarning			: ST_IO2_SingleInputCtrl:=			(eTypeInput:=E_IO2_Type.NO,		tTimeOnFilter:=t#10ms, 		tTimeOffFilter:=t#0ms, 	sInputName:='Labeller2 Summar yWarning' );	(**)
	st_I_Labeller2Error							: ST_IO2_SingleInputCtrl:=			(eTypeInput:=E_IO2_Type.NO,		tTimeOnFilter:=t#10ms, 		tTimeOffFilter:=t#0ms, 	sInputName:='Labeller2 Error' );	(**)

(*METS SADDLE (Gating&Reject System) Filtered Inputs  FB***************************************************************************************************************)
	st_I_OuterAtClamp					: ST_IO2_SingleInputCtrl:=			(eTypeInput:=E_IO2_Type.NO,		tTimeOnFilter:=t#100ms, 		tTimeOffFilter:=t#100ms, 		sInputName:='Outer At Clamp');	(**)
	st_I_OuterAtLabelGate				: ST_IO2_SingleInputCtrl:=			(eTypeInput:=E_IO2_Type.NO,		tTimeOnFilter:=t#100ms, 		tTimeOffFilter:=t#100ms, 		sInputName:='Outer At Label Gate');	(**)
	st_I_GateClear						: ST_IO2_SingleInputCtrl:=			(eTypeInput:=E_IO2_Type.NO,		tTimeOnFilter:=t#100ms, 		tTimeOffFilter:=t#100ms, 		sInputName:='Gate Clear');	(**)
	st_I_GateImpact					: ST_IO2_SingleInputCtrl:=			(eTypeInput:=E_IO2_Type.NO,		tTimeOnFilter:=t#100ms, 		tTimeOffFilter:=t#100ms, 		sInputName:='Gate Impact');	(**)

(* Single Inputs for METS CML*)
	st_I_RotaryTransferPackAtStopPlate		: ST_IO2_SingleInputCtrl:=			(eTypeInput:=E_IO2_Type.NO,		tTimeOnFilter:=t#1000ms, 		tTimeOffFilter:=t#0ms, 	sInputName:='Rotary Transfer Outer At Stop Plate');	(**)
	st_I_RotaryTransferTorqueLimiter			: ST_IO2_SingleInputCtrl:=			(eTypeInput:=E_IO2_Type.NO,		tTimeOnFilter:=t#1000ms, 		tTimeOffFilter:=t#0ms, 	sInputName:='Rotary Transfer Torque Limiter');	(**)
	st_I_RotaryTransferDelayStop1			: ST_IO2_SingleInputCtrl:=			(eTypeInput:=E_IO2_Type.NO,		tTimeOnFilter:=t#1000ms, 		tTimeOffFilter:=t#0ms, 	sInputName:='Rotary Transfer Delay Stop1');	(**)
	st_I_RotaryTransferDelayStop2			: ST_IO2_SingleInputCtrl:=			(eTypeInput:=E_IO2_Type.NO,		tTimeOnFilter:=t#1000ms, 		tTimeOffFilter:=t#0ms, 	sInputName:='Rotary Transfer Delay Stop2');	(**)
	st_I_ConveyorIndexContact				: ST_IO2_SingleInputCtrl:=			(eTypeInput:=E_IO2_Type.NO,		tTimeOnFilter:=t#50ms, 		tTimeOffFilter:=t#50s, 	sInputName:='Infeed Conveyor Start');	(**)
	st_I_Guard4ElectricalBoxInPosition		: ST_IO2_SingleInputCtrl:=			(eTypeInput:=E_IO2_Type.NC,		tTimeOnFilter:=t#50ms, 		tTimeOffFilter:=t#50s, 	sInputName:='Electrical Box In Position Sensor');	(**)

(* Single Inputs for METS Manual Machine*)
	st_I_InfeedConveyorStart				: ST_IO2_SingleInputCtrl:=			(eTypeInput:=E_IO2_Type.NO,		tTimeOnFilter:=t#1000ms, 		tTimeOffFilter:=t#0ms, 	sInputName:='Infeed Conveyor Start');	(**)
	st_I_RejectChuteExitBlocked			: ST_IO2_SingleInputCtrl:=			(eTypeInput:=E_IO2_Type.NO,		tTimeOnFilter:=t#1000ms, 		tTimeOffFilter:=t#0ms, 	sInputName:='Reject Chute Blocked');	(**)

(* Single Inputs for METS SFLX Machine*)
	st_I_OuterInfeedJam						: ST_IO2_SingleInputCtrl:=			(eTypeInput:=E_IO2_Type.NO,		tTimeOnFilter:=t#1000ms, 		tTimeOffFilter:=t#0ms, 	sInputName:='Outer Infeed Jam' );	(**)
	(*st_I_PackAggregationCameraTrigger		: ST_IO2_SingleInputCtrl:=			(eTypeInput:=E_IO2_Type.NO,		tTimeOnFilter:=t#1000ms, 		tTimeOffFilter:=t#0ms, 	sInputName:='Pack Aggregation Camera Trigger');*)	(**)
	st_I_OutfeedConveyorStart				: ST_IO2_SingleInputCtrl:=			(eTypeInput:=E_IO2_Type.NO,		tTimeOnFilter:=t#1000ms, 		tTimeOffFilter:=t#0ms, 	sInputName:='Outfeed Conveyor Start');	(**)
	st_I_RejectConfirmationNCW				: ST_IO2_SingleInputCtrl:=			(eTypeInput:=E_IO2_Type.NO,		tTimeOnFilter:=t#1000ms, 		tTimeOffFilter:=t#0ms, 	sInputName:='Reject Confirmation NCW');	(**)
	st_I_RejectBinFullNCW						: ST_IO2_SingleInputCtrl:=			(eTypeInput:=E_IO2_Type.NO,		tTimeOnFilter:=t#1000ms, 		tTimeOffFilter:=t#0ms, 	sInputName:='Reject Bin Full NCW');	(**)
	st_I_OuterAtTransferReject				: ST_IO2_SingleInputCtrl:=			(eTypeInput:=E_IO2_Type.NO,		tTimeOnFilter:=t#1000ms, 		tTimeOffFilter:=t#0ms, 	sInputName:='Outer At Transfer Reject');	(**)
	st_I_OuterAtSideFlexExit					: ST_IO2_SingleInputCtrl:=			(eTypeInput:=E_IO2_Type.NO,		tTimeOnFilter:=t#1000ms, 		tTimeOffFilter:=t#0ms, 	sInputName:='Outer At Side Flex Exit');	(**)
	st_I_OuterAtPostMachineInfeed			: ST_IO2_SingleInputCtrl:=			(eTypeInput:=E_IO2_Type.NO,		tTimeOnFilter:=t#1000ms, 		tTimeOffFilter:=t#0ms, 	sInputName:='Outer At PostMachine Infeed');	(**)

	st_I_Guard1FlexInfeedDoor				: ST_IO2_SingleInputCtrl:=			(eTypeInput:=E_IO2_Type.NC,		tTimeOnFilter:=t#1000ms, 		tTimeOffFilter:=t#0ms, 	sInputName:='Guard 1 Flex Infeed Door');	(**)
	st_I_Guard3FlexRHDoor					: ST_IO2_SingleInputCtrl:=			(eTypeInput:=E_IO2_Type.NO,		tTimeOnFilter:=t#200ms, 		tTimeOffFilter:=t#200ms, 	sInputName:='Guard 3 Flex RH Door');	(**)
	st_I_Guard4FlexPrinterDoor				: ST_IO2_SingleInputCtrl:=			(eTypeInput:=E_IO2_Type.NO,		tTimeOnFilter:=t#200ms, 		tTimeOffFilter:=t#200ms, 	sInputName:='Guard 4 Flex Printer Door');	(**)
	st_I_Guard5FlexLHDoor					: ST_IO2_SingleInputCtrl:=			(eTypeInput:=E_IO2_Type.NO,		tTimeOnFilter:=t#200ms, 		tTimeOffFilter:=t#200ms, 	sInputName:='Guard 5 Flex LH Door	');	(**)

(*Single Input for PACAN*)
(*	st_I_StackerArmAtBackwardPosition	: ST_IO2_SingleInputCtrl:=			(eTypeInput:=E_IO2_Type.NO,		tTimeOnFilter:=t#10ms, 		tTimeOffFilter:=t#0ms, 	sInputName:='Stacker Arm At Backward Position');	(**)
	st_I_StackerArmInTopPosition			: ST_IO2_SingleInputCtrl:=			(eTypeInput:=E_IO2_Type.NO,		tTimeOnFilter:=t#10ms, 		tTimeOffFilter:=t#0ms, 	sInputName:='Stacker Arm In Top Position');	(**)
	st_I_StackPresentSensor1				: ST_IO2_SingleInputCtrl:=			(eTypeInput:=E_IO2_Type.NO,		tTimeOnFilter:=t#10ms, 		tTimeOffFilter:=t#0ms, 	sInputName:='Stack Present Sensor1');	(**)
	st_I_StackPresentSensor2				: ST_IO2_SingleInputCtrl:=			(eTypeInput:=E_IO2_Type.NO,		tTimeOnFilter:=t#10ms, 		tTimeOffFilter:=t#0ms, 	sInputName:='Stack Present Sensor2');	(**)
	st_I_StackerTransferPusher			: ST_IO2_SingleInputCtrl:=			(eTypeInput:=E_IO2_Type.NO,		tTimeOnFilter:=t#10ms, 		tTimeOffFilter:=t#0ms, 	sInputName:='Stacker Transfer Pusher');	(**)
	st_I_StackerTransferComplete			: ST_IO2_SingleInputCtrl:=			(eTypeInput:=E_IO2_Type.NO,		tTimeOnFilter:=t#10ms, 		tTimeOffFilter:=t#0ms, 	sInputName:='Stacker Transfer Complete');	(**)
	st_I_OuterAtPACANRejectStation		: ST_IO2_SingleInputCtrl:=			(eTypeInput:=E_IO2_Type.NO,		tTimeOnFilter:=t#100ms, 		tTimeOffFilter:=t#100ms, 	sInputName:='Outer At PACAN Reject Station');	(**)
*)
(*Single Input for PAOL*)
	st_I_TPDExitBlockedSensor			: ST_IO2_SingleInputCtrl:=			(eTypeInput:=E_IO2_Type.NO,		tTimeOnFilter:=t#100ms, 		tTimeOffFilter:=t#0ms, 	sInputName:='PAOL Exit Blocked Sensor');	(**)
	st_I_PreMachineBuildBackSensor		: ST_IO2_SingleInputCtrl:=			(eTypeInput:=E_IO2_Type.NO,		tTimeOnFilter:=t#100ms, 		tTimeOffFilter:=t#0ms, 	sInputName:='PAOL Buildback Sensor');	(**)
	st_I_PackAggregCameraRigSensor		: ST_IO2_SingleInputCtrl:=			(eTypeInput:=E_IO2_Type.NO,		tTimeOnFilter:=t#6ms, 		tTimeOffFilter:=t#6ms, 	sInputName:='Pack Aggreg Camera Rig Sensor');	(**)

(*Single Input for PLAS*)
	st_I_MasterlistDoorGuard1				: ST_IO2_SingleInputCtrl:=			(eTypeInput:=E_IO2_Type.NC,		tTimeOnFilter:=t#50ms, 		tTimeOffFilter:=t#50ms, 	sInputName:='Masterlist Door Guard1');	(**)
	st_I_MasterlistDoorGuard2				: ST_IO2_SingleInputCtrl:=			(eTypeInput:=E_IO2_Type.NC,		tTimeOnFilter:=t#50ms, 		tTimeOffFilter:=t#50ms, 	sInputName:='Masterlist Door Guard2');	(**)
	st_I_MasterlistDoorGuard3				: ST_IO2_SingleInputCtrl:=			(eTypeInput:=E_IO2_Type.NC,		tTimeOnFilter:=t#50ms, 		tTimeOffFilter:=t#50ms, 	sInputName:='Masterlist Door Guard3');	(**)

	st_I_OuterBrushOpen						: ST_IO2_SingleInputCtrl:=			(eTypeInput:=E_IO2_Type.NC,		tTimeOnFilter:=t#50ms, 		tTimeOffFilter:=t#50ms, 	sInputName:='Outer Brush Open');	(**)
	st_I_PackAggregationDoorGuard1			: ST_IO2_SingleInputCtrl:=			(eTypeInput:=E_IO2_Type.NC,		tTimeOnFilter:=t#50ms, 		tTimeOffFilter:=t#50ms, 	sInputName:='Pack Aggregation Door Guard1');	(**)
	st_I_PackAggregationDoorGuard2			: ST_IO2_SingleInputCtrl:=			(eTypeInput:=E_IO2_Type.NC,		tTimeOnFilter:=t#50ms, 		tTimeOffFilter:=t#50ms, 	sInputName:='Pack Aggregation Door Guard2');	(**)

	st_I_WrapperDoorGuard1					:  ST_IO2_SingleInputCtrl:=			(eTypeInput:=E_IO2_Type.NC,		tTimeOnFilter:=t#50ms, 		tTimeOffFilter:=t#50ms, 	sInputName:='Wrapper Door Guard1');	(**)
	st_I_WrapperDoorGuard2					: ST_IO2_SingleInputCtrl:=			(eTypeInput:=E_IO2_Type.NC,		tTimeOnFilter:=t#50ms, 		tTimeOffFilter:=t#50ms, 	sInputName:='Wrapper Door Guard2');	(**)

	st_I_HeatTunelPackReject				: ST_IO2_SingleInputCtrl:=			(eTypeInput:=E_IO2_Type.NO,		tTimeOnFilter:=t#50ms, 		tTimeOffFilter:=t#50ms, 	sInputName:='Heat Tunenel Pack Reject Sensor');	(**)
	st_I_WrapperPackReject				: ST_IO2_SingleInputCtrl:=			(eTypeInput:=E_IO2_Type.NC,		tTimeOnFilter:=t#50ms, 		tTimeOffFilter:=t#50ms, 	sInputName:='Wrapper Pack Reject Sensor');	(**)
	st_I_WrapperPackReject2				: ST_IO2_SingleInputCtrl:=			(eTypeInput:=E_IO2_Type.NC,		tTimeOnFilter:=t#50ms, 		tTimeOffFilter:=t#50ms, 	sInputName:='Wrapper Pack Reject 2 Sensor');	(**)
	st_I_WrapperOuterComplete			: ST_IO2_SingleInputCtrl:=			(eTypeInput:=E_IO2_Type.NC,		tTimeOnFilter:=t#50ms, 		tTimeOffFilter:=t#50ms, 	sInputName:='Wrapper Pushing Arm Sensor');	(**)
	st_I_InhibitIntermediateCamera		: ST_IO2_SingleInputCtrl:=			(eTypeInput:=E_IO2_Type.NC,		tTimeOnFilter:=t#50ms, 		tTimeOffFilter:=t#50ms, 	sInputName:='Inhibit Intermediate Camera');	(**)

(*Single Input for Laser*)
	st_I_CoderReady					: ST_IO2_SingleInputCtrl:=			(eTypeInput:=E_IO2_Type.NO,		tTimeOnFilter:=t#100ms, 		tTimeOffFilter:=t#0ms, 	sInputName:='LASER - Ready');	(**)
	st_I_CoderBusy					: ST_IO2_SingleInputCtrl:=			(eTypeInput:=E_IO2_Type.NO,		tTimeOnFilter:=t#100ms, 		tTimeOffFilter:=t#0ms, 	sInputName:='LASER - Busy');	(**)
	st_I_WrappingMaterialPresent		: ST_IO2_SingleInputCtrl:=			(eTypeInput:=E_IO2_Type.NO,		tTimeOnFilter:=t#100ms, 		tTimeOffFilter:=t#0ms, 	sInputName:='LASER - WrapPresent');	(**)
	st_I_TabKnifeMoving				: ST_IO2_SingleInputCtrl:=			(eTypeInput:=E_IO2_Type.NO,		tTimeOnFilter:=t#100ms, 		tTimeOffFilter:=t#0ms, 	sInputName:='LASER - TabKnife');	(**)


(*******************************************************************************************************************************************************)
(********************************************************Double IO******************************************************************************)
(*******************************************************************************************************************************************************)
(*Double Input Config*)
	st_I_RowComplete						: ST_IO2_DoubleInputCtrl:=		(eInputSource:=E_IO2_InputSource.SENSOR,	sInputName:='Row Complete',
																						eTypeInput1:=E_IO2_Type.NO,		tTimeOnFilter1:=t#0ms,	tTimeOffFilter1	:=t#0ms,	(**)
											 											eTypeInput2:=E_IO2_Type.NO,		tTimeOnFilter2:=t#0ms,	tTimeOffFilter2	:=t#0ms);	(**)
	st_I_LayerComplete					: ST_IO2_DoubleInputCtrl:=		(eInputSource:=E_IO2_InputSource.SENSOR,	sInputName:='Layer Complete',
																						eTypeInput1:=E_IO2_Type.NO,		tTimeOnFilter1:=t#0ms,	tTimeOffFilter1	:=t#0ms,	(**)
											 											eTypeInput2:=E_IO2_Type.NO,		tTimeOnFilter2:=t#0ms,	tTimeOffFilter2	:=t#0ms);	(**)
	st_I_IntermediatePush					: ST_IO2_DoubleInputCtrl:=		(eInputSource:=E_IO2_InputSource.SENSOR,	sInputName:='Intermediate Push',
																						eTypeInput1:=E_IO2_Type.NO,		tTimeOnFilter1:=t#0ms,	tTimeOffFilter1	:=t#0ms,	(**)
											 											eTypeInput2:=E_IO2_Type.NO,		tTimeOnFilter2:=t#0ms,	tTimeOffFilter2	:=t#0ms);	(**)
	st_I_CaseComplete					: ST_IO2_DoubleInputCtrl:=		(eInputSource:=E_IO2_InputSource.SENSOR,	sInputName:='Case Complete',
																						eTypeInput1:=E_IO2_Type.NO,		tTimeOnFilter1:=t#0ms,	tTimeOffFilter1	:=t#0ms,	(**)
											 											eTypeInput2:=E_IO2_Type.NO,		tTimeOnFilter2:=t#0ms,	tTimeOffFilter2	:=t#0ms);	(**)
	st_I_CaseDischarged					: ST_IO2_DoubleInputCtrl:=		(eInputSource:=E_IO2_InputSource.SENSOR,	sInputName:='Case Discharged',
																						eTypeInput1:=E_IO2_Type.NO,		tTimeOnFilter1:=t#0ms,	tTimeOffFilter1	:=t#0ms,	(**)
											 											eTypeInput2:=E_IO2_Type.NO,		tTimeOnFilter2:=t#0ms,	tTimeOffFilter2	:=t#0ms);	(**)
	st_I_CaseLabelValidation				: ST_IO2_DoubleInputCtrl:=		(eInputSource:=E_IO2_InputSource.SENSOR,	sInputName:='Case Label Validation',
																						eTypeInput1:=E_IO2_Type.NO,		tTimeOnFilter1:=t#0ms,	tTimeOffFilter1	:=t#0ms,	(**)
											 											eTypeInput2:=E_IO2_Type.NO,		tTimeOnFilter2:=t#0ms,	tTimeOffFilter2	:=t#0ms);	(**)
(*
	st_I_LiftComplete						: ST_IO2_DoubleInputCtrl:=		(eInputSource:=SENSOR,		eTypeInput1:=E_IO2_Type.NO,		tTimeOnFilter1:=t#0ms,	tTimeOffFilter1	:=t#0ms,	(**)
											 											eTypeInput2:=E_IO2_Type.NO,		tTimeOnFilter2:=t#0ms,	tTimeOffFilter2	:=t#0ms);	(**)
	st_I_StackComplete					: ST_IO2_DoubleInputCtrl:=		(eInputSource:=SENSOR,		eTypeInput1:=E_IO2_Type.NO,		tTimeOnFilter1:=t#0ms,	tTimeOffFilter1	:=t#0ms,	(**)
											 											eTypeInput2:=E_IO2_Type.NO,		tTimeOnFilter2:=t#0ms,	tTimeOffFilter2	:=t#0ms);	(**)
	st_I_BundleCrossPushComplete		: ST_IO2_DoubleInputCtrl:=		(eInputSource:=SENSOR,		eTypeInput1:=E_IO2_Type.NO,		tTimeOnFilter1:=t#0ms,	tTimeOffFilter1	:=t#0ms,	(**)
											 											eTypeInput2:=E_IO2_Type.NO,		tTimeOnFilter2:=t#0ms,	tTimeOffFilter2	:=t#0ms);	(**)
	st_I_BundleTranferComplete			: ST_IO2_DoubleInputCtrl:=		(eInputSource:=SENSOR,		eTypeInput1:=E_IO2_Type.NO,		tTimeOnFilter1:=t#0ms,	tTimeOffFilter1	:=t#0ms,	(**)
											 											eTypeInput2:=E_IO2_Type.NO,		tTimeOnFilter2:=t#0ms,	tTimeOffFilter2	:=t#0ms);	(**)
*)

(*******************************************************************************************************************************************************)
(********************************************************Outpurs******************************************************************************)
(*******************************************************************************************************************************************************)
(*Output Config*)
	st_Q_TPDMachineRun					: ST_IO2_OutputCtrl:=			(eTypeOutput:=E_IO2_Type.NO,		tOutputDelayed:=t#0ms,		tOutputLocked:=t#0ms,	sOutputName:='TPD Machine Run');		(* *)
	st_Q_CMLConvoyerRun				: ST_IO2_OutputCtrl:=			(eTypeOutput:=E_IO2_Type.NO,		tOutputDelayed:=t#0ms,		tOutputLocked:=t#0ms,	sOutputName:='CML Convoyer Run');		(* *)
	st_Q_EUCAPreMachineRun				: ST_IO2_OutputCtrl:=			(eTypeOutput:=E_IO2_Type.NO,		tOutputDelayed:=t#0ms,		tOutputLocked:=t#0ms,	sOutputName:='EUCA Machine Run');		(* *)
	st_Q_EUCAMachineRun				: ST_IO2_OutputCtrl:=			(eTypeOutput:=E_IO2_Type.NO,		tOutputDelayed:=t#0ms,		tOutputLocked:=t#0ms,	sOutputName:='EUCA Machine Run');		(* *)
	st_Q_CaseContentOK					: ST_IO2_OutputCtrl:=			(eTypeOutput:=E_IO2_Type.NO,		tOutputDelayed:=t#0ms,		tOutputLocked:=t#0ms,	sOutputName:='Case Content OK');		(* *)
	st_Q_CaseValidationOK				: ST_IO2_OutputCtrl:=			(eTypeOutput:=E_IO2_Type.NO,		tOutputDelayed:=t#0ms,		tOutputLocked:=t#0ms,	sOutputName:='Case Validation OK');		(* *)
	st_Q_OuterValidationOK				: ST_IO2_OutputCtrl:=			(eTypeOutput:=E_IO2_Type.NO,		tOutputDelayed:=t#0ms,		tOutputLocked:=t#0ms,	sOutputName:='Outer Validation OK');		(* *)
	st_Q_LabellerInhibit					: ST_IO2_OutputCtrl:=			(eTypeOutput:=E_IO2_Type.NO,		tOutputDelayed:=t#0ms,		tOutputLocked:=t#0ms,	sOutputName:='Labeller Inhibit');		(* *)
	st_Q_SideBeltDriveBrake				: ST_IO2_OutputCtrl:=			(eTypeOutput:=E_IO2_Type.NO,		tOutputDelayed:=t#500ms,	tOutputLocked:=t#20ms,	sOutputName:='Side Belt Drive Brake');		(* *)
	st_Q_PackSeparatorDriveBrake			: ST_IO2_OutputCtrl:=			(eTypeOutput:=E_IO2_Type.NO,		tOutputDelayed:=t#200ms,	tOutputLocked:=t#100ms,sOutputName:='Pack Separator Drive Brake');		(* *)

	st_Q_CameraLightning1				: ST_IO2_OutputCtrl:=			(eTypeOutput:=E_IO2_Type.NO,		tOutputDelayed:=t#0ms,		tOutputLocked:=t#15ms,	sOutputName:='Camera Lightning 1');		(* *)
	st_Q_CameraLightning2				: ST_IO2_OutputCtrl:=			(eTypeOutput:=E_IO2_Type.NO,		tOutputDelayed:=t#0ms,		tOutputLocked:=t#15ms,	sOutputName:='Camera Lightning 2');		(* *)
	st_Q_CameraLightning3				: ST_IO2_OutputCtrl:=			(eTypeOutput:=E_IO2_Type.NO,		tOutputDelayed:=t#0ms,		tOutputLocked:=t#15ms,	sOutputName:='Camera Lightning 3');		(* *)
	st_Q_CameraLightning4				: ST_IO2_OutputCtrl:=			(eTypeOutput:=E_IO2_Type.NO,		tOutputDelayed:=t#0ms,		tOutputLocked:=t#15ms,	sOutputName:='Camera Lightning 4');		(* *)
	st_Q_CameraLightning5				: ST_IO2_OutputCtrl:=			(eTypeOutput:=E_IO2_Type.NO,		tOutputDelayed:=t#0ms,		tOutputLocked:=t#15ms,	sOutputName:='Camera Lightning 5');		(* *)
	st_Q_CameraLightning6				: ST_IO2_OutputCtrl:=			(eTypeOutput:=E_IO2_Type.NO,		tOutputDelayed:=t#0ms,		tOutputLocked:=t#15ms,	sOutputName:='Camera Lightning 6');		(* *)
	st_Q_CameraLightning7				: ST_IO2_OutputCtrl:=			(eTypeOutput:=E_IO2_Type.NO,		tOutputDelayed:=t#0ms,		tOutputLocked:=t#15ms,	sOutputName:='Camera Lightning 7');		(* *)
	st_Q_CameraLightning8				: ST_IO2_OutputCtrl:=			(eTypeOutput:=E_IO2_Type.NO,		tOutputDelayed:=t#0ms,		tOutputLocked:=t#15ms,	sOutputName:='Camera Lightning 8');		(* *)
	st_Q_CameraLightning9				: ST_IO2_OutputCtrl:=			(eTypeOutput:=E_IO2_Type.NO,		tOutputDelayed:=t#0ms,		tOutputLocked:=t#15ms,	sOutputName:='Camera Lightning 9');		(* *)
	st_Q_CameraLightning10				: ST_IO2_OutputCtrl:=			(eTypeOutput:=E_IO2_Type.NO,		tOutputDelayed:=t#0ms,		tOutputLocked:=t#15ms,	sOutputName:='Camera Lightning 10');	(* *)
	st_Q_CameraLightning11				: ST_IO2_OutputCtrl:=			(eTypeOutput:=E_IO2_Type.NO,		tOutputDelayed:=t#0ms,		tOutputLocked:=t#15ms,	sOutputName:='Camera Lightning 11');	(* *)
	st_Q_CameraLightning12				: ST_IO2_OutputCtrl:=			(eTypeOutput:=E_IO2_Type.NO,		tOutputDelayed:=t#0ms,		tOutputLocked:=t#15ms,	sOutputName:='Camera Lightning 12');	(* *)

(*Output Config for camera triggers*)
(*
	st_Q_Camera01						: ST_IO2_OutputCtrl:=			(eTypeOutput:=E_IO2_Type.NO,		tOutputDelayed:=t#0ms,		tOutputLocked:=t#0ms);		(* *)
	st_Q_Camera02						: ST_IO2_OutputCtrl:=			(eTypeOutput:=E_IO2_Type.NO,		tOutputDelayed:=t#0ms,		tOutputLocked:=t#0ms);		(* *)
	st_Q_Camera03						: ST_IO2_OutputCtrl:=			(eTypeOutput:=E_IO2_Type.NO,		tOutputDelayed:=t#0ms,		tOutputLocked:=t#0ms);		(* *)
	st_Q_Camera04						: ST_IO2_OutputCtrl:=			(eTypeOutput:=E_IO2_Type.NO,		tOutputDelayed:=t#0ms,		tOutputLocked:=t#0ms);		(* *)
	st_Q_Camera05						: ST_IO2_OutputCtrl:=			(eTypeOutput:=E_IO2_Type.NO,		tOutputDelayed:=t#0ms,		tOutputLocked:=t#0ms);		(* *)
	st_Q_Camera06						: ST_IO2_OutputCtrl:=			(eTypeOutput:=E_IO2_Type.NO,		tOutputDelayed:=t#0ms,		tOutputLocked:=t#0ms);		(* *)
	st_Q_Camera07						: ST_IO2_OutputCtrl:=			(eTypeOutput:=E_IO2_Type.NO,		tOutputDelayed:=t#0ms,		tOutputLocked:=t#0ms);		(* *)
	st_Q_Camera08						: ST_IO2_OutputCtrl:=			(eTypeOutput:=E_IO2_Type.NO,		tOutputDelayed:=t#0ms,		tOutputLocked:=t#0ms);		(* *)
	st_Q_Camera09						: ST_IO2_OutputCtrl:=			(eTypeOutput:=E_IO2_Type.NO,		tOutputDelayed:=t#0ms,		tOutputLocked:=t#0ms);		(* *)
	st_Q_Camera10						: ST_IO2_OutputCtrl:=			(eTypeOutput:=E_IO2_Type.NO,		tOutputDelayed:=t#0ms,		tOutputLocked:=t#0ms);		(* *)
	st_Q_Camera11						: ST_IO2_OutputCtrl:=			(eTypeOutput:=E_IO2_Type.NO,		tOutputDelayed:=t#0ms,		tOutputLocked:=t#0ms);		(* *)
	st_Q_Camera12						: ST_IO2_OutputCtrl:=			(eTypeOutput:=E_IO2_Type.NO,		tOutputDelayed:=t#0ms,		tOutputLocked:=t#0ms);		(* *)
*)
END_STRUCT
END_TYPE

// ---- DUTs/METS/System/ST_SYSTEM_DateTime.TcDUT
TYPE ST_SYSTEM_DateTime :
STRUCT
	bSystemTimeValid		: BOOL;
	sSystemTime			: TIMESTRUCT;
	nSystemTimeOffset		: DINT;			(* sSystemTime offset from UTC in ms *)
	sUTCTime				: TIMESTRUCT;
	sUTCTimeZoneOffset	: STRING(6);		(*Time Zone Offset from HMI in ISO 8601 format*)
	sOffsetTime			: TIMESTRUCT;
	bPCMTimeValid		: BOOL;
	sPCMTime			: TIMESTRUCT;
	strHMIDateTime		: STRING(19);	(* date/time as HH:MM:SS DD/MM/YYYY for HMI display *)
END_STRUCT
END_TYPE

// ---- DUTs/METS/System/ST_SYSTEM_DeviceState.TcDUT
TYPE ST_SYSTEM_DeviceState :
STRUCT
	aCameraIPSettingsValid	: ARRAY[1..cMAX_CAMERA_NUMBER] OF BOOL;
	aCameraStatus			: ARRAY[1..cMAX_CAMERA_NUMBER] OF ST_SCANNER;	(**)

	aHandScannersValid		: ARRAY[1..cMAX_HAND_SCANNERS] OF BOOL;
	aHandScanners			: ARRAY[0..cMAX_HAND_SCANNERS] OF ST_SCANNER_HoneywellStatus;		(* index 0 used for DigitalTwin input*)
	aHandScannerHostAck	: ARRAY[1..cMAX_HAND_SCANNERS] OF ST_SCANNER_HostAck;			(**)

	aPrinterIPSettingsValid	: ARRAY[1..cMAX_PRINTER_NUMBER] OF BOOL;
	aPrinterStatus			: ARRAY[1..cMAX_PRINTER_NUMBER] OF ST_PRINTER_Status;	(**)

	aDriverStatus			: ARRAY[1..cMAX_ANALOG_DRIVERS] OF ST_DriveCtrl;
	aPNetMasterStatus		: ARRAY [1..cMAX_PROFINET_MASTERS]  OF  ST_PNetMasterStatus;
	aDriveInterfaces		: ARRAY[1..cMAX_PROFINET_DRIVES] OF ST_G120_Status;
	aMC2AxisStatus		: ARRAY[1..cMAX_MC2_DRIVES] OF ST_AXIS_Status;

	(*aAFS50CamStatus		: ARRAY [1..cMAX_CAMS] OF ST_AFS60_Status;*)
	aEncoderStatus		: ARRAY[1..cMAX_ENCODER] OF ST_ENCODER_Status;

	aCylinderStatus		: ARRAY[1..cMAX_CYLINDERS] OF ST_CYLINDER_Status;

END_STRUCT
END_TYPE

// ---- DUTs/METS/System/ST_SYSTEM_Door.TcDUT
TYPE ST_SYSTEM_Door :
STRUCT
	bClearConveyorQueue						: BOOL;
	bClearPackerQueue							: BOOL;
	aClearCaseQueue							: ARRAY[1..cMAX_CASE_QUEUE] OF BOOL;
END_STRUCT
END_TYPE

// ---- DUTs/METS/System/ST_SYSTEM_MachineMode.TcDUT
TYPE ST_SYSTEM_MachineMode :
STRUCT
	bDisable			: BOOL;
	bManual			: BOOL;
	bAutomatic		:  BOOL;
END_STRUCT
END_TYPE

// ---- DUTs/METS/System/ST_SYSTEM_MachineState.TcDUT
TYPE ST_SYSTEM_MachineState :
STRUCT

	bSystemPowerUp 				: BOOL;
	bImmediateStopped 			: BOOL;
	bMachineInError				: BOOL;
	bSystemInitialising 			: BOOL;
	bManualMode					: BOOL;
	bSystemReadyToStart 			: BOOL;
	bSystemCycleStopping			: BOOL;
	bSystemRunning				: BOOL;
	bMachineWaitingForProduct	: BOOL;
	bMachineInConditionalRun	: BOOL;
	bTrackAndTraceDeactivated	: BOOL;
END_STRUCT
END_TYPE

// ---- DUTs/METS/System/ST_SYSTEM_ProductionLine.TcDUT
TYPE ST_SYSTEM_ProductionLine :
STRUCT
	sPCM			: STRING(4);
	sMENo			: STRING(5);
	nTopologyID	: INT;
END_STRUCT
END_TYPE

// ---- DUTs/METS/System/ST_SYSTEM_SafetyStatus.TcDUT
TYPE ST_SYSTEM_SafetyStatus :
STRUCT
	bSafetyRelayOK					: BOOL;
	bEStopButtonPressed				: BOOL;
	bEmergencyCircuitOK				: BOOL;
	bGuardDoorOK						: BOOL;
	bMotorDriversOK					: BOOL;
	bSafetyOK						: BOOL;			(* All systems Go! *)

END_STRUCT
END_TYPE

// ---- DUTs/METS/System/ST_SYSTEM_SoftwareVersion.TcDUT
TYPE ST_SYSTEM_SoftwareVersion :
STRUCT
	sPLCVersionHMI					: STRING;
	sScreenVersionInfoHMI				: STRING;
	sBridgeVersionHMI					: STRING;
END_STRUCT
END_TYPE

// ---- DUTs/METS/System/System Modes/E_SYSTEM_PackAggregationMode.TcDUT
//{attribute 'strict'}
TYPE E_SYSTEM_PackAggregationMode :
(
	E_SYSTEM_NOPACKAGGREGATION		:= 0,
	E_SYSTEM_PAOL_2CAM				:= 1,
	E_SYSTEM_PAOL_3CAM				:= 2,
	E_SYSTEM_PLAS_T01					:= 3,		(*GD, 2cam linear, clearwrap*)
	E_SYSTEM_PLAS_T02					:= 4,	(*GD, 2 cam, preprint outer label  -> until no info in PCM about production, this include into FB_PCM_Validate*)
	E_SYSTEM_PLAS_T03					:= 5,		(*FOCKE multistack, single type production*)
	E_SYSTEM_PLAS_T04					:= 6		(* FOCKE HYBRID NON CLEAR WRAP - Validation as confirmation *)
);
END_TYPE

// ---- DUTs/METS/TCPIP Address/E_TCPIP_State_1.TcDUT
TYPE E_TCPIP_State_1 :
(
	E_TCPIP_IDLE,
	E_TCPIP_CONNECT,
	E_TCPIP_SEND,
	E_TCPIP_RECEIVE,
	E_TCPIP_DISCONNECT,
	E_TCPIP_CLOSEALL,
	E_TCPIP_DONE
);
END_TYPE

// ---- DUTs/METS/TCPIP Address/ST_TCPIP_AddressPort.TcDUT
TYPE ST_TCPIP_AddressPort :
STRUCT
	IP			: T_IPv4Addr;
	Port		: UINT;
END_STRUCT
END_TYPE

// ---- DUTs/METS/XML Processing/E_XML_CtrlState.TcDUT
TYPE E_XML_CtrlState :
(
	E_XML_IDLE,
	E_XML_COPYTOCURRENT,
	E_XML_READXML,
	E_XML_VALIDATE,
	E_XML_GENERATEIMAGE,
	E_XML_WRITEXML,
	E_XML_CHECKFILESIZE,
	E_XML_DONE
);
END_TYPE

// ---- DUTs/METS/XML Processing/E_XML_GeneratorState.TcDUT
TYPE E_XML_GeneratorState :
(
	E_XML_GENERATOR_IDLE,
	E_XML_GENERATE_HEAD_CHM,
	E_XML_DONE_HEAD_CHM,
	E_XML_GENERATE_BODY_CHM,
	E_XML_DONE_BODY_CHM,
	E_XML_GENERATE_ENDING_CHM,
	E_XML_DONE_ENDING_CHM,
	E_XML_GENERATE_GMES,
	E_XML_DONE_GMES,
	E_XML_GENERATE_FLG,
	E_XML_DONE_FLG,
	E_XML_GENERATE_GMES_FLG,
	E_XML_DONE_GMES_FLG,
	E_XML_GENERATOR_DONE
);
END_TYPE

// ---- DUTs/METS/XML Processing/E_XML_WritingMode.TcDUT
TYPE E_XML_WritingMode :
(
	E_CS_HEADER,
	E_OUTER_HEADER,
	E_PACK_ITEM,
	E_OUTER_ENDING,
	E_CS_ENDING
);
END_TYPE

// ---- DUTs/METS/_StationOperational/C715 Tempalate Example/E_04_ElevatorState_C715.TcDUT
TYPE E_04_ElevatorState_C715 :
(
	SEQ_04_INIT									:=0,
	SEQ_04_ENABLEDEVICES							:=1,
	SEQ_04_HOMING								:=10,
	SEQ_04_MOVETODOWNLIMIT_DONE				:=20,
	SEQ_04_HOMINGWITHDATUM						:=30,

	SEQ_04_MOVETOHOMEPOS_TRY					:=40,
	SEQ_04_MOVETOHOMEPOS_DONE					:=50,
	SEQ_04_HOMED								:=90,
	SEQ_04_READY									:=100,

	SEQ_04_REQACCEPTED							:=110,

	SEQ_04_MOVEUP_TRY							:=120,
	SEQ_04_MOVEUP_DONE							:=130,
	SEQ_04_UNLOADBUNDLE_TRY						:=140,
	SEQ_04_UNLOADBUNDLE_DONE					:=150,

	SEQ_04_MOVEPOSITIVE_TRY						:=160,
	SEQ_04_MOVEPOSITIVE_DONE						:=170,
	SEQ_04_MOVENEGATIVE_TRY						:=180,
	SEQ_04_MOVENEGATIVE_DONE					:=190,
	SEQ_04_REJECTEXTEND_TRY						:=200,
	SEQ_04_REJECTEXTEND_DONE						:=210,
	SEQ_04_REJECTRETRACT_TRY						:=220,
	SEQ_04_REJECTRETRACT_DONE						:=230,


	(*SEQ_04_MOVEDOWN_TRY						:=160,
	SEQ_04_MOVEDOWN_DONE						:=170,*)

	SEQ_04_COMPLETE_TRY							:=340,
	SEQ_04_COMPLETE								:=350

);
END_TYPE

// ---- DUTs/METS/_StationOperational/C715 Tempalate Example/E_Axis_C715.TcDUT
TYPE E_Axis_C715 :
(
	E_C715_WALKINGBEAM	:=1,
	E_C715_ELEVATOR		:=2,
	E_C715_TRANSFER		:=3,
	E_C715_PRESENTATION	:=4

);
END_TYPE

// ---- DUTs/METS/_StationOperational/C715 Tempalate Example/E_Cylinder_C715.TcDUT
TYPE E_Cylinder_C715 :
(
	E_C715_STOPGATE01		:=1,
	E_C715_STOPGATE02		:=2,
	E_C715_BUNDLEALIGN	:=3,
	E_C715_TAMPHEAD		:=4,
	E_C715_LABELFORM		:=5,
	E_C715_BUNDLEREJECT	:=6,
	E_C715_BUNDLEPUSH	:=7

);
END_TYPE

// ---- DUTs/METS/_StationOperational/C715 Tempalate Example/ST_04_ElevatorSeq_C715.TcDUT
  TYPE ST_04_ElevatorSeq_C715 :
STRUCT
	e04SeqState					: E_04_ElevatorState_C715;

